(* CODESYS project IndraLogic.project

Project tree, tasks and I/O mapping:
  IndraMotionMlc1 : IndraControl XM2, Bosch Rexroth AG, order no. dependent on customer specific configuration, version 14.18.31.0
    application Application
      libraries: ML_TechBase, 14.18.0.0 (System); VisuDialogs, * (System)
      task SCC_Task (externalevent, external event EVENT_OP_MODE_MOTION_CYCLIC, priority 3, watchdog 1000 µs x 2) calls SCC, VCC, HMI
      task Acc_Sensor_Task (cyclic, interval t#2ms, priority 6) calls Acc_Sensor
      function CheckBounds [ST]
      global variables GV
      Symbols
      program VCC [FBD]
      program SCC [FBD]
      global variables MlcVarGlobal
      trace Trace (task MotionTask): VCC_Testing.uPF
      global variables UDP_Send
      function block VCC_StepFunction_Test [ST]
      trace Controller (task MotionTask): UDP_Send.Vel_RefGen, UDP_Send.Pos_RefGen, UDP_Send.nRef
      function block StepFunction_Test_Christian [ST]
      function block Input_Signals [FBD]
      function block Real_Time_Counter [FBD]
      function block Enable_Motion_SCC [FBD]
      function block JoyStick_SCC [FBD]
      function block LoadHolding_Control [FBD]
      function block JoyStick_VCC [FBD]
      function block Enable_Motion_VCC [FBD]
      function block VCC_PI_Controller [ST]
      program HMI [FBD]
      function block CyclSercosChnl [FBD]
      function block SinuousCurve_Test [ST]
      function block Ramp_Test [ST]
      function block CC_PI_FF_AD [ST]
      program VCC_Controller [FBD]
      function block VCC_Joystick_vel_ref [FBD]
      function block FIR_FIlter [ST]
      function block Discrete_FIlter [ST]
      program VCC_Testing [FBD]
      function block SCC_Controller [FBD]
      program VCC_Anti_DB [FBD]
      function block VCC_Anti_Dead_Band_v2 [ST]
      function block Subsystem [ST]
      function block VCC_SP_Ramp_Generator [ST]
      function block VCC_Controller_FF_PI_AD [ST]
      function block S_shape_Profile_old [ST]
      function block Ramp_Profile [ST]
      function block SCC_Controller_FF_PI_AD [ST]
      function block VCC_Controller_FF_PI_AD_v04 [ST]
      function block VCC_Controller_FF_PI_AD_v05 [ST]
      program VCC_PRV_Control [FBD]
      function block VCC_PRV_Mapping [ST]
      function block Discrete_Lowpass_Filter0 [ST]
      function block VCC_PV_Controller [ST]
      function block VCC_StepFunction [ST]
      function block VCC_Step_Function_Validation [ST]
      function block PF2 [ST]
      function block PF1 [ST]
      function block SCC_LPPF [ST]
      function block HPPF_pB [ST]
      function block HPPF2_pB [ST]
      function block HPPF_pA [ST]
      function block HPPF2_pA [ST]
      function block VCC_Controller_PI_FF [ST]
      function block Step_Damiano [ST]
      function block SCC_Ramp_Test [ST]
      function block SCC_HPPF [ST]
      function block SCC_DPF [ST]
      function block ZCFCN_d_FALLING [ST]
      function block ZCFCN_d_ANY [ST]
      function block SCC_Controller_VFF [ST]
      function block SCC_Controller_PFB [ST]
      function block Low_Pass_Filter [ST]
      function block SCC_PFB_Controller_PID [ST]
      function block SCC_PFB_Controller_PID2 [ST]
      function block SCC_SinProfile [ST]
      function block CascadedControllerFilter [ST]
      function block LHV_Controller [ST]
      function block LHV_Enabler [ST]
      function block Pressure_Feed_Forward [ST]
      function block SCC_Controller_PFB1 [ST]
      function block SCC_Vel_AD [ST]
      function block SCC_VFF [ST]
      function block SCC_HPPF1 [ST]
      function block LHV_Controller2 [ST]
      function block Delay_Vel [ST]
      function block Delay_Pos [ST]
      function block VCC_Controller_PFB [ST]
      function block VCC_VFF [ST]
      function block VCC_Pos_Step [ST]
      function block SCC_AD_Iq [ST]
      function block S_shape_Profile [ST]
      global variables UDP_Send_Acc
      program Acc_Sensor [FBD]
      function block SCC_Secondary_Controller [FBD]
      function block SCC_Primary_Controller [FBD]
      function block Primary_Control2 [ST]
      function block Primary_Control1 [ST]
      function block Primary_Control3 [ST]
      function block Secondary_Control [ST]
      function block LPF [ST]
      function block JoyStick_SCC_TrqCntrl [FBD]
      Visualization/
        SCC/
          visualisation SCC
          SubWindows/
            visualisation SCC_Main
            visualisation SCC_activeDamping
        VCC/
          visualisation VCC_Visualization
          visualisation VCC_Filtered_LS
          SubWindows/
      function block SCC_Acceleration_Feedback [ST]
    S20_I_O : S20_I_O, Bosch Rexroth AG, version 14.18.20.0
      S20_AI_8 : S20-AI-8, Bosch Rexroth AG, order no. R911172536, version Revision=16#0
          settings: Analog Input.IDN = 16#010005E1; Analog Input.IDN = 16#010005E1; PropritaryParameterSet_P-1-0128.0.0.IDN = 16#01009080; PropritaryParameterSet_P-1-0128.0.0.Abort if error = False; PropritaryParameterSet_P-1-0128.0.0.Jump to line if error = False; PropritaryParameterSet_P-1-0128.0.0.SercosAttribute = 16#00000000
          input  CylPos : WORD  // Analog Input.Analog Input 1
          input  p1 : WORD  // Analog Input.Analog Input 2
          input  p2 : WORD  // Analog Input.Analog Input 3
          input  p3 : WORD  // Analog Input.Analog Input 4
          input  p4 : WORD  // Analog Input.Analog Input 5
          input  p5 : WORD  // Analog Input.Analog Input 6
          input  p6 : WORD  // Analog Input.Analog Input 7
          input  p7 : WORD  // Analog Input.Analog Input 8
          unmapped channels: Analog Input
      S20_AI_8_1 : S20-AI-8, Bosch Rexroth AG, order no. R911172536, version Revision=16#0
          settings: Analog Input.IDN = 16#010005E1; Analog Input.IDN = 16#010005E1; PropritaryParameterSet_P-1-0128.0.0.IDN = 16#01009080; PropritaryParameterSet_P-1-0128.0.0.Abort if error = False; PropritaryParameterSet_P-1-0128.0.0.Jump to line if error = False; PropritaryParameterSet_P-1-0128.0.0.SercosAttribute = 16#00000000
          input  p8 : WORD  // Analog Input.Analog Input 1
          input  p9 : WORD  // Analog Input.Analog Input 2
          input  p10 : WORD  // Analog Input.Analog Input 3
          input  p11 : WORD  // Analog Input.Analog Input 4
          input  T11 : WORD  // Analog Input.Analog Input 5
          input  T6 : WORD  // Analog Input.Analog Input 6
          input  T4 : WORD  // Analog Input.Analog Input 7
          input  Acc_Y_raw : WORD  // Analog Input.Analog Input 8
          unmapped channels: Analog Input
      S20_AI_8_2 : S20-AI-8, Bosch Rexroth AG, order no. R911172536, version Revision=16#0
          settings: Analog Input.IDN = 16#010005E1; Analog Input.IDN = 16#010005E1; PropritaryParameterSet_P-1-0128.0.0.IDN = 16#01009080; PropritaryParameterSet_P-1-0128.0.0.Abort if error = False; PropritaryParameterSet_P-1-0128.0.0.Jump to line if error = False; PropritaryParameterSet_P-1-0128.0.0.SercosAttribute = 16#00000000
          input  p_pump : WORD  // Analog Input.Analog Input 1
          input  p_return : WORD  // Analog Input.Analog Input 2
          input  p_compensator : WORD  // Analog Input.Analog Input 3
          input  p_A : WORD  // Analog Input.Analog Input 4
          input  p_A1 : WORD  // Analog Input.Analog Input 5
          input  p_B : WORD  // Analog Input.Analog Input 6
          input  Q_B : WORD  // Analog Input.Analog Input 7
          input  JoyY : WORD  // Analog Input.Analog Input 8
          unmapped channels: Analog Input
      S20_AI6_AO2_SSI2 : S20-AI6-AO2-SSI2, Bosch Rexroth AG, order no. R911173120, version Revision=16#0
          settings: Analog Output.IDN = 16#010005E0; Analog Input.IDN = 16#010005E1; Positioning.IDN = 16#010005EB; Analog Output.IDN = 16#010005E0; Analog Input.IDN = 16#010005E1; Positioning.IDN = 16#010005EB; PropritaryParameterSet_P-1-0041.0.0.IDN = 16#01009029; PropritaryParameterSet_P-1-0041.0.0.Abort if error = False; PropritaryParameterSet_P-1-0041.0.0.Jump to line if error = False; PropritaryParameterSet_P-1-0041.0.0.SercosAttribute = 16#00000000; PropritaryParameterSet_P-1-0128.0.0.IDN = 16#01009080; PropritaryParameterSet_P-1-0128.0.0.Abort if error = False; PropritaryParameterSet_P-1-0128.0.0.Jump to line if error = False; PropritaryParameterSet_P-1-0128.0.0.SercosAttribute = 16#00000000; PropritaryParameterSet_P-1-0128.0.0 = [16#02,16#00,16#02,16#00,16#05,16#05]; PropritaryParameterSet_S-0-1504.0.2.IDN = 16#010205E0; PropritaryParameterSet_S-0-1504.0.2.Abort if error = False; PropritaryParameterSet_S-0-1504.0.2.Jump to line if error = False; PropritaryParameterSet_S-0-1504.0.2.SercosAttribute = 16#00000000; PropritaryParameterSet_P-1-0047.0.0.IDN = 16#0100902F; PropritaryParameterSet_P-1-0047.0.0.Abort if error = False; PropritaryParameterSet_P-1-0047.0.0.Jump to line if error = False; PropritaryParameterSet_P-1-0047.0.0.SercosAttribute = 16#00000000; PropritaryParameterSet_P-1-0128.0.1.IDN = 16#01019080; PropritaryParameterSet_P-1-0128.0.1.Abort if error = False; PropritaryParameterSet_P-1-0128.0.1.Jump to line if error = False; PropritaryParameterSet_P-1-0128.0.1.SercosAttribute = 16#00000000; PropritaryParameterSet_P-1-0128.0.1 = [16#0C,16#00,16#0C,16#00,16#05,16#05,16#0F,16#00,16#00,16#00,16#0F,16#0F,16#0F,16#00,16#00,16#00]; PropritaryParameterSet_P-1-0128.0.2.IDN = 16#01029080; PropritaryParameterSet_P-1-0128.0.2.Abort if error = False; PropritaryParameterSet_P-1-0128.0.2.Jump to line if error = False; PropritaryParameterSet_P-1-0128.0.2.SercosAttribute = 16#00000000; PropritaryParameterSet_P-1-0128.0.3.IDN = 16#01039080; PropritaryParameterSet_P-1-0128.0.3.Abort if error = False; PropritaryParameterSet_P-1-0128.0.3.Jump to line if error = False; PropritaryParameterSet_P-1-0128.0.3.SercosAttribute = 16#00000000; PropritaryParameterSet_P-1-0129.0.0.IDN = 16#01009081; PropritaryParameterSet_P-1-0129.0.0.Abort if error = False; PropritaryParameterSet_P-1-0129.0.0.Jump to line if error = False; PropritaryParameterSet_P-1-0129.0.0.SercosAttribute = 16#00000000;
            PropritaryParameterSet_P-1-0129.0.1.IDN = 16#01019081; PropritaryParameterSet_P-1-0129.0.1.Abort if error = False; PropritaryParameterSet_P-1-0129.0.1.Jump to line if error = False; PropritaryParameterSet_P-1-0129.0.1.SercosAttribute = 16#00000000; PropritaryParameterSet_P-1-0041.0.0.IDN = 16#01009029; PropritaryParameterSet_P-1-0041.0.0.Abort if error = False; PropritaryParameterSet_P-1-0041.0.0.Jump to line if error = False; PropritaryParameterSet_P-1-0041.0.0.SercosAttribute = 16#00000000
          output PVG_Us : WORD  // Analog Output.Analog Output 1
          output PRV_Cmd : WORD  // Analog Output.Analog Output 2
          input  PVG_SP : WORD  // Analog Input.Analog Input1
          input  PRV_Act : WORD  // Analog Input.Analog Input2
          unmapped channels: Analog Output, Analog Input, Positioning
      S20_DI_16_4 : S20-DI-16/4, Bosch Rexroth AG, order no. R911172532, version Revision=16#0
          settings: Digital Input.IDN = 16#010005DF; Digital Input.IDN = 16#010005DF; PropritaryParameterSet_S-0-1503.0.20.IDN = 16#011405DF
          input  startBtn : BOOL  // Digital Input.Digital Input Byte 0.00
          input  stopBtn : BOOL  // Digital Input.Digital Input Byte 0.01
          input  manMode : BOOL  // Digital Input.Digital Input Byte 0.02
          input  autoMode : BOOL  // Digital Input.Digital Input Byte 0.03
          unmapped channels: Digital Input
      S20_DO_16_3 : S20-DO-16/3, Bosch Rexroth AG, order no. R911172534, version Revision=16#0
          settings: Digital Output.IDN = 16#010005DE; Digital Output.IDN = 16#010005DE; PropritaryParameterSet_S-0-1502.0.2.IDN = 16#010205DE; PropritaryParameterSet_S-0-1502.0.20.IDN = 16#011405DE
          output LHvalve : BOOL  // Digital Output.Digital Output Byte 0.00
          output Motion_Start_Light : BOOL  // Digital Output.Digital Output Byte 0.01
          output Motion_Stop_Light : BOOL  // Digital Output.Digital Output Byte 0.02
          output CoolerFan : BOOL  // Digital Output.Digital Output Byte 0.03
          output PVG_Udc : BOOL  // Digital Output.Digital Output Byte 0.04
          unmapped channels: Digital Output
    Sercos_III_Master : SercosIII Master, Rexroth, order no. 1, version 14.6.0.0
    RT_Ethernet_Slave_XFE01_1_FB_04 : RT-Ethernet Slave(XFE01.1-FB-04), Bosch Rexroth AG, order no. R911173937, version 14.14.0.0
      Not_Used : Not Used, Bosch Rexroth AG, version 14.8.0.0
    EtherNet_IP_Adapter_on_Eng_Port : EtherNet/IP Adapter on Eng.-Port, Bosch Rexroth AG, version 12.10.2.0
      _8_Byte_Input : 8 Byte Input, Bosch Rexroth AG, version 12.10.2.0
          unmapped channels: Channel1
      _8_Byte_Output_4Byte_Run_Header : 8 Byte Output + 4Byte Run Header, Bosch Rexroth AG, version 12.10.2.0
          unmapped channels: Channel1
  libraries: VisuSymbols, 3.5.8.0 (System)
  text list GlobalTextList
*)

// IndraMotionMlc1/Application/GV

VAR_GLOBAL
	TestMode: BOOL;

	UDP_ON: BOOL;
	SCC_ON: BOOL := 0;
	SCC_On_Light: BOOL;
	SCC_ManModeVelAct: BOOL;
	SCC_AutoModeVelAct: BOOL;
	SCC_Motion_Stop_Light: BOOL;
	SCC_Manual_Mode_Enable: BOOL;
	SCC_Manual_Max_Speed: REAL := 1000.0;
	SCC_Auto_Mode_Enable: BOOL;
	SCC_Control_Mode: BOOL := 0;
	SCC_Control_Mode_Enabled: BOOL;
	SCC_Cntrl_Error_Limit: LREAL := 1;
	SCC_Cntrl_s0: LREAL := 50.0;
	SCC_Cntrl_tHold_Up_Up_Up: LREAL:= 5.0;
	SCC_Cntrl_t0: LREAL := 5.0;
	SCC_Cntrl_Pos_SP: LREAL := 200.0;
	SCC_Cntrl_Vel_SP: LREAL := 50.0;
	SCC_Cntrl_k_P: LREAL := 2.7227E+04;
	SCC_Cntrl_T_I: LREAL := 3.4851E+04;
	SCC_Cntrl_k_P_AD: LREAL := 1.4125E+05;
	SCC_Cntrl_T_I_AD: LREAL := 1.2204E+05;
	SCC_Tuning_Mode: BOOL := 0;
	SCC_S_shape_On: BOOL :=1;
	SCC_Vel_Ref_Max: REAL := 120;
	SCC_k_AD: LREAL := 2.112E-11 ;
	SCC_tau_AD: LREAL := 0.993;
	SCC_Cntrl_Motion_Cycle_Time: LREAL;
    SCC_Test_Mode: BOOL := 0; 
	SCC_Test_Mode_Enabled: BOOL := 0; 
	SCC_FB_Cntr_On: BOOL;
	SCC_FB_Cntr_Enabled: BOOL;
	SCC_I_Cntr_On: BOOL :=0;
	SCC_AD_On: BOOL :=0;
	SCC_LH_Valve_Activated: BOOL; 
	SCC_Passive_LH_On: BOOL; 
	SCC_Cntrl_FF_On: BOOL := 1;
	SCC_Cntrl_FF_up: LREAL := 1.6450e-07;
    SCC_Cntrl_FF_down: LREAL := 1.7500E-07;
	SCC_Vel_RefGen: LREAL; 
	SCC_Pos_RefGen: LREAL; 
	SCC_RecordTime: LREAL; 
	SCC_vel_AD_On: BOOL:= 0;
	SCC_vel_AD_kf: LREAL:= 1.995E04;
	SCC_vel_AD_tauf: LREAL:= 0.9934;
	SCC_HPPF_On: BOOL:= 0;
	SCC_HPPF_Reset: BOOL:= 0;
	SCC_HPPF_kf: LREAL:= 4.239E-11;
	SCC_HPPF_tauf: LREAL:= 0.999;
	SCC_LPPF_On: BOOL:= 0;
	SCC_LPPF_kf: LREAL:= 1.223E-12; 
	SCC_LPPF_tauf: LREAL:= 0.9737;
	SCC_DPF_On: BOOL:= 0;
	SCC_DPF_kf: LREAL:= 3.7255E-11;
	Joystick_Ref: LREAL; 
	SCC_OL_On: BOOL:= 0;
	SCC_Sin_Test_On: BOOL := 0;
    SCC_SinTest_T: LREAL:= 10;
	SCC_Motor_ON: BOOL := 0;
	SCC_Force_Motor_ON: BOOL := 0;
	
	SCC_LHV_OFF: BOOL := 0;
	SCC_LHV_ON: BOOL := 0;
	
	SCC_PosError_limit: LREAL:= 0.5;
	
	SCC_LHC_On: BOOL := 0;
	SCC_LHC_FF_On: BOOL := 1;
	SCC_LHC_kP: LREAL:= 0.000015;
	SCC_LHC_FF_kP: LREAL:= 0.000015;
	SCC_LHC_error_SP: LREAL:= 1;
	SCC_LHC_vel_lim: LREAL:= 0.1;
	SCC_LHC_openingDelay: TIME:= T#200MS;
	SCC_LHC_openingDelay2: TIME:= T#5MS;
	SCC_LHC_openingDelay3: TIME:= T#3S;
	SCC_Delay_ms: LREAL:= 100; 
	SCC_LHC_nSP: LREAL:= 300;
	Pos_Ref_Delay: LREAL;
	Vel_Ref_Delay: LREAL;
	Pos_Ref_Act: LREAL;
	Vel_Ref_Act: LREAL;
	SCC_Motion_Delay_On: BOOL := 0;
    SCC_Step_Test_On: BOOL := 0; 
    Mode_Selected: BOOL;
	
	SCC_AD_Iq_On: BOOL:= 0;
	SCC_k_AD_Iq: LREAL := 0 ;
	
	// Secondary Controller
	SCC_Enable_TCTR : BOOL:= 0; 
	SCC_SCTR_ON : BOOL:= 0; 
    SCC_AutoModeTorqueAct: BOOL; 
	
	// Acceleration Feedback (AF)
	SCC_AF_On: BOOL := 0;
	SCC_AF_Direct_On : BOOL := 0;
	SCC_AF_LPF_On : BOOL := 0;
	SCC_AF_LPF_w : BOOL := 0;
	SCC_AF_HPF_On : BOOL := 0;

	SCC_AF_Acc_Input_raw : LREAL;
	SCC_AF_Acc_Input : LREAL;
	SCC_AF_Acc_Input_DB : LREAL := 0.1;
	
	SCC_AF_D_rev : LREAL := 10.6;
	SCC_AF_K_direct : LREAL := 1.7045E-04;
	SCC_AF_LPF_Num1 : LREAL := 0;
	SCC_AF_LPF_Num2 : LREAL := 1.39E-05;
	SCC_AF_LPF_Den1 : LREAL := 1;
	SCC_AF_LPF_Den2 : LREAL := -0.9418;
	SCC_AF_HPF_Num1 : LREAL := 2.6846E-04;
	SCC_AF_HPF_Num2 : LREAL := -2.6846E-04;
	SCC_AF_HPF_Den1 : LREAL := 1;
	SCC_AF_HPF_Den2 : LREAL := -0.9955;

	Ramp_tHold: LREAL:= 1;
	Ramp_tWait: LREAL:= 1;
	tRamp: LREAL:= 1;
	nSP: LREAL:= 1000;
	
	VCC_ON: BOOL := 0; 
	VCC_On_Light: BOOL;
	VCC_Manual_Mode_Enabled: BOOL; 
	VCC_S_shape_On: BOOL :=1;
    VCC_Vel_Ref_Max: REAL := 120;
    VCC_Max_Joy_Output: REAL := 100.0;
    VCC_Auto_Mode_Enabled: BOOL; 
	VCC_Control_Mode: BOOL := 0;
    VCC_Control_Mode_Enabled: BOOL := 0;
	VCC_FB_Cntr_On: BOOL :=0;
	VCC_FB_Cntr_Enabled: BOOL;
	VCC_I_Cntr_On: BOOL :=0;
	VCC_AD_On: BOOL :=0;
	VCC_k_AD: LREAL := 0.004;
	VCC_Cntrl_DB_up: LREAL := 0.114;
	VCC_Cntrl_Motion_Cycle_Time: LREAL;
    VCC_Cntrl_DB_down: LREAL := 0.13;
	VCC_Cntrl_Error_Limit: LREAL := 1;
	VCC_Cntrl_s0: LREAL := 50.0;
	VCC_Cntrl_Trvl_Dist: LREAL := 200.0;
	VCC_Cntrl_tHold: LREAL:= 5.0;
	VCC_Cntrl_t0: LREAL := 3.0;
	VCC_Cntrl_Vel_SP: LREAL := 50.0;
	VCC_Cntrl_k_P: LREAL := 29.1743;
	VCC_Cntrl_T_I: LREAL := 19.4884;
	VCC_Tuning_Mode: BOOL := 0;
	VCC_Test_Mode: BOOL := 0; 
	VCC_Test_Mode_Enabled: BOOL := 0; 
	VCC_Ramp_Test_On: BOOL := 0; 
	VCC_Ramp_Test_u_DCV_1: LREAL := 0; 
	VCC_Ramp_Test_u_DCV_2: LREAL := 0; 
	VCC_Ramp_Test_tR: LREAL := 1; 
	VCC_Ramp_Test_tHold_Up: LREAL := 5; 
	VCC_Ramp_Test_tHold_Down: LREAL := 5; 
	VCC_Ramp_Test_tWait: LREAL := 5; 
	VCC_Step_Test_On: BOOL := 0; 
	VCC_Step_Test_t0: LREAL := 1;
	VCC_Step_Test_tWait: LREAL := 1;
	VCC_Step_Test_tWait2: LREAL := 1;
    VCC_Step_Test_tStepUp: LREAL := 1;
	VCC_Step_Test_tStepDown: LREAL := 1;
	VCC_Step_Test_SP: LREAL := 0.1;
	VCC_Step_Test_u0: LREAL := 0.05;
	VCC_Step_Test_Up: BOOL := 0; 
	VCC_Sin_Test_On: BOOL := 0; 
	VCC_Test_t0: LREAL := 1.0;
	VCC_Vel_RefGen: LREAL; 
	VCC_Pos_RefGen: LREAL; 
	VCC_RecordTime: LREAL; 
	VCC_Cntrl_Q_max_up: LREAL := 30.0;
	VCC_Cntrl_Q_max_down: LREAL := 30.0;
	VCC_Cntrl_FF_Valve_Mapping_On: BOOL := 0; 
	VCC_Cntrl_Integral_Reset_On: BOOL := 1; 
	VCC_PRV_Cntrl_p_C_Max: LREAL := 75; 
	VCC_PRV_Cntrl_p_C_Min: LREAL := 4; 
	VCC_PRV_Cntrl_Opening: LREAL := 0;
	VCC_PRV_Cntrl_Opening_SP: LREAL := 0;
	VCC_PRV_Cntrl_Enable: BOOL := 0;
	VCC_PRV_Cntrl_Enabled: BOOL;
	VCC_PRV_Cntrl_Auto_On: BOOL := 0;
	VCC_PRV_p_C_SP: LREAL := 0;
	VCC_PRV_Cntrl_Manual_Pressure_On: BOOL;
	VCC_PRV_Cntrl_k_LPF: LREAL :=1;
	VCC_PRV_Cntrl_T_LPF: LREAL :=0.5;
	VCC_PRV_Cntrl_k_P: LREAL := 1; 
	VCC_PRV_Cntrl_T_I: LREAL := 0; 
	VCC_PRV_Cntrl_FF_On: BOOL := 1; 
	VCC_PRV_Cntrl_LPF_On: BOOL := 1; 
	VCC_PRV_Cntrl_Tuning_Mode_On: BOOL := 0; 
	VCC_PF2_On: BOOL := 0; 
	VCC_PF1_On: BOOL := 0; 
    VCC_PF_pB_On: BOOL := 0; 
	VCC_PF_pB_vInv_On: BOOL := 0; 
	VCC_PF_pA_vInv_On: BOOL := 0; 
	VCC_PF_pL_vInv_On: BOOL := 0; 
	VCC_PF_Test_On: BOOL := 0; 
	VCC_PF_HP_Num1: LREAL := 1.176E-11;  
	VCC_PF_HP_Den1: LREAL := 1;
	VCC_PF_HP_Den2: LREAL := -0.9957;
	VCC_PF1_HP_Num1: LREAL := 9.019E-12;  
	VCC_PF1_HP_Den1: LREAL := 1;
	VCC_PF1_HP_Den2: LREAL := -0.9905;
	VCC_PF_pB_HP_Num1: LREAL := 1.344E-11;  
	VCC_PF_pB_HP_Den1: LREAL := 1;
	VCC_PF_pB_HP_Den2: LREAL := -0.9951;
	VCC_PF_ADB_On: BOOL := 0; 
	VCC_LPPF_On: BOOL := 0; 
	VCC_LPPF_Num1: LREAL := 8.647E-13;  
	VCC_LPPF_Den1: LREAL := 1;
	VCC_LPPF_Den2: LREAL := -0.8424;
	VCC_SinTest_freq: LREAL := 0;
	VCC_SinTest_Amp: LREAL := 0;
	VCC_Cntrl_uPF: LREAL := 0;
END_VAR

// IndraMotionMlc1/Application/MlcVarGlobal
(* Automatically generated code by XLC/MLC. *)
(* Please don't edit, the code will be overwritten. For usercode use UserVarGlobal! *)
{attribute 'linkalways'}
{attribute 'analysis' := '-33'}
VAR_GLOBAL CONSTANT

(*LREAL axis "Drive1" with axis number 1*)
Drive1: AXIS_REF :=(CntrlNo:=LOCAL_CNTRL,AxisNo:=AXIS_1);


(*Probe 001*)
TouchProbe001: TOUCHPROBE_REF :=(CntrlNo:=LOCAL_CNTRL,TouchProbeNo:=TOUCHPROBE_1);

(*Probe 002*)
TouchProbe002: TOUCHPROBE_REF :=(CntrlNo:=LOCAL_CNTRL,TouchProbeNo:=TOUCHPROBE_2);

(*Probe 003*)
TouchProbe003: TOUCHPROBE_REF :=(CntrlNo:=LOCAL_CNTRL,TouchProbeNo:=TOUCHPROBE_3);

(*Probe 004*)
TouchProbe004: TOUCHPROBE_REF :=(CntrlNo:=LOCAL_CNTRL,TouchProbeNo:=TOUCHPROBE_4);

(*Probe 005*)
TouchProbe005: TOUCHPROBE_REF :=(CntrlNo:=LOCAL_CNTRL,TouchProbeNo:=TOUCHPROBE_5);

(*Probe 006*)
TouchProbe006: TOUCHPROBE_REF :=(CntrlNo:=LOCAL_CNTRL,TouchProbeNo:=TOUCHPROBE_6);

(*Probe 007*)
TouchProbe007: TOUCHPROBE_REF :=(CntrlNo:=LOCAL_CNTRL,TouchProbeNo:=TOUCHPROBE_7);

(*Probe 008*)
TouchProbe008: TOUCHPROBE_REF :=(CntrlNo:=LOCAL_CNTRL,TouchProbeNo:=TOUCHPROBE_8);

(*Probe 009*)
TouchProbe009: TOUCHPROBE_REF :=(CntrlNo:=LOCAL_CNTRL,TouchProbeNo:=TOUCHPROBE_9);

(*Probe 010*)
TouchProbe010: TOUCHPROBE_REF :=(CntrlNo:=LOCAL_CNTRL,TouchProbeNo:=TOUCHPROBE_10);

(*Probe 011*)
TouchProbe011: TOUCHPROBE_REF :=(CntrlNo:=LOCAL_CNTRL,TouchProbeNo:=TOUCHPROBE_11);

(*Probe 012*)
TouchProbe012: TOUCHPROBE_REF :=(CntrlNo:=LOCAL_CNTRL,TouchProbeNo:=TOUCHPROBE_12);

(*Probe 013*)
TouchProbe013: TOUCHPROBE_REF :=(CntrlNo:=LOCAL_CNTRL,TouchProbeNo:=TOUCHPROBE_13);

(*Probe 014*)
TouchProbe014: TOUCHPROBE_REF :=(CntrlNo:=LOCAL_CNTRL,TouchProbeNo:=TOUCHPROBE_14);

(*Probe 015*)
TouchProbe015: TOUCHPROBE_REF :=(CntrlNo:=LOCAL_CNTRL,TouchProbeNo:=TOUCHPROBE_15);

(*Probe 016*)
TouchProbe016: TOUCHPROBE_REF :=(CntrlNo:=LOCAL_CNTRL,TouchProbeNo:=TOUCHPROBE_16);

(*Probe 017*)
TouchProbe017: TOUCHPROBE_REF :=(CntrlNo:=LOCAL_CNTRL,TouchProbeNo:=TOUCHPROBE_17);

(*Probe 018*)
TouchProbe018: TOUCHPROBE_REF :=(CntrlNo:=LOCAL_CNTRL,TouchProbeNo:=TOUCHPROBE_18);

(*Probe 019*)
TouchProbe019: TOUCHPROBE_REF :=(CntrlNo:=LOCAL_CNTRL,TouchProbeNo:=TOUCHPROBE_19);

(*Probe 020*)
TouchProbe020: TOUCHPROBE_REF :=(CntrlNo:=LOCAL_CNTRL,TouchProbeNo:=TOUCHPROBE_20);

(*Probe 021*)
TouchProbe021: TOUCHPROBE_REF :=(CntrlNo:=LOCAL_CNTRL,TouchProbeNo:=TOUCHPROBE_21);

(*Probe 022*)
TouchProbe022: TOUCHPROBE_REF :=(CntrlNo:=LOCAL_CNTRL,TouchProbeNo:=TOUCHPROBE_22);

(*Probe 023*)
TouchProbe023: TOUCHPROBE_REF :=(CntrlNo:=LOCAL_CNTRL,TouchProbeNo:=TOUCHPROBE_23);

(*Probe 024*)
TouchProbe024: TOUCHPROBE_REF :=(CntrlNo:=LOCAL_CNTRL,TouchProbeNo:=TOUCHPROBE_24);

(*Probe 025*)
TouchProbe025: TOUCHPROBE_REF :=(CntrlNo:=LOCAL_CNTRL,TouchProbeNo:=TOUCHPROBE_25);

(*Probe 026*)
TouchProbe026: TOUCHPROBE_REF :=(CntrlNo:=LOCAL_CNTRL,TouchProbeNo:=TOUCHPROBE_26);

(*Probe 027*)
TouchProbe027: TOUCHPROBE_REF :=(CntrlNo:=LOCAL_CNTRL,TouchProbeNo:=TOUCHPROBE_27);

(*Probe 028*)
TouchProbe028: TOUCHPROBE_REF :=(CntrlNo:=LOCAL_CNTRL,TouchProbeNo:=TOUCHPROBE_28);

(*Probe 029*)
TouchProbe029: TOUCHPROBE_REF :=(CntrlNo:=LOCAL_CNTRL,TouchProbeNo:=TOUCHPROBE_29);

(*Probe 030*)
TouchProbe030: TOUCHPROBE_REF :=(CntrlNo:=LOCAL_CNTRL,TouchProbeNo:=TOUCHPROBE_30);

(*Probe 031*)
TouchProbe031: TOUCHPROBE_REF :=(CntrlNo:=LOCAL_CNTRL,TouchProbeNo:=TOUCHPROBE_31);

(*Probe 032*)
TouchProbe032: TOUCHPROBE_REF :=(CntrlNo:=LOCAL_CNTRL,TouchProbeNo:=TOUCHPROBE_32);

(*Probe 033*)
TouchProbe033: TOUCHPROBE_REF :=(CntrlNo:=LOCAL_CNTRL,TouchProbeNo:=TOUCHPROBE_33);

(*Probe 034*)
TouchProbe034: TOUCHPROBE_REF :=(CntrlNo:=LOCAL_CNTRL,TouchProbeNo:=TOUCHPROBE_34);

(*Probe 035*)
TouchProbe035: TOUCHPROBE_REF :=(CntrlNo:=LOCAL_CNTRL,TouchProbeNo:=TOUCHPROBE_35);

(*Probe 036*)
TouchProbe036: TOUCHPROBE_REF :=(CntrlNo:=LOCAL_CNTRL,TouchProbeNo:=TOUCHPROBE_36);

(*Probe 037*)
TouchProbe037: TOUCHPROBE_REF :=(CntrlNo:=LOCAL_CNTRL,TouchProbeNo:=TOUCHPROBE_37);

(*Probe 038*)
TouchProbe038: TOUCHPROBE_REF :=(CntrlNo:=LOCAL_CNTRL,TouchProbeNo:=TOUCHPROBE_38);

(*Probe 039*)
TouchProbe039: TOUCHPROBE_REF :=(CntrlNo:=LOCAL_CNTRL,TouchProbeNo:=TOUCHPROBE_39);

(*Probe 040*)
TouchProbe040: TOUCHPROBE_REF :=(CntrlNo:=LOCAL_CNTRL,TouchProbeNo:=TOUCHPROBE_40);

(*Probe 041*)
TouchProbe041: TOUCHPROBE_REF :=(CntrlNo:=LOCAL_CNTRL,TouchProbeNo:=TOUCHPROBE_41);

(*Probe 042*)
TouchProbe042: TOUCHPROBE_REF :=(CntrlNo:=LOCAL_CNTRL,TouchProbeNo:=TOUCHPROBE_42);

(*Probe 043*)
TouchProbe043: TOUCHPROBE_REF :=(CntrlNo:=LOCAL_CNTRL,TouchProbeNo:=TOUCHPROBE_43);

(*Probe 044*)
TouchProbe044: TOUCHPROBE_REF :=(CntrlNo:=LOCAL_CNTRL,TouchProbeNo:=TOUCHPROBE_44);

(*Probe 045*)
TouchProbe045: TOUCHPROBE_REF :=(CntrlNo:=LOCAL_CNTRL,TouchProbeNo:=TOUCHPROBE_45);

(*Probe 046*)
TouchProbe046: TOUCHPROBE_REF :=(CntrlNo:=LOCAL_CNTRL,TouchProbeNo:=TOUCHPROBE_46);

(*Probe 047*)
TouchProbe047: TOUCHPROBE_REF :=(CntrlNo:=LOCAL_CNTRL,TouchProbeNo:=TOUCHPROBE_47);

(*Probe 048*)
TouchProbe048: TOUCHPROBE_REF :=(CntrlNo:=LOCAL_CNTRL,TouchProbeNo:=TOUCHPROBE_48);

(*Probe 049*)
TouchProbe049: TOUCHPROBE_REF :=(CntrlNo:=LOCAL_CNTRL,TouchProbeNo:=TOUCHPROBE_49);

(*Probe 050*)
TouchProbe050: TOUCHPROBE_REF :=(CntrlNo:=LOCAL_CNTRL,TouchProbeNo:=TOUCHPROBE_50);

(*Probe 051*)
TouchProbe051: TOUCHPROBE_REF :=(CntrlNo:=LOCAL_CNTRL,TouchProbeNo:=TOUCHPROBE_51);

(*Probe 052*)
TouchProbe052: TOUCHPROBE_REF :=(CntrlNo:=LOCAL_CNTRL,TouchProbeNo:=TOUCHPROBE_52);

(*Probe 053*)
TouchProbe053: TOUCHPROBE_REF :=(CntrlNo:=LOCAL_CNTRL,TouchProbeNo:=TOUCHPROBE_53);

(*Probe 054*)
TouchProbe054: TOUCHPROBE_REF :=(CntrlNo:=LOCAL_CNTRL,TouchProbeNo:=TOUCHPROBE_54);

(*Probe 055*)
TouchProbe055: TOUCHPROBE_REF :=(CntrlNo:=LOCAL_CNTRL,TouchProbeNo:=TOUCHPROBE_55);

(*Probe 056*)
TouchProbe056: TOUCHPROBE_REF :=(CntrlNo:=LOCAL_CNTRL,TouchProbeNo:=TOUCHPROBE_56);

(*Probe 057*)
TouchProbe057: TOUCHPROBE_REF :=(CntrlNo:=LOCAL_CNTRL,TouchProbeNo:=TOUCHPROBE_57);

(*Probe 058*)
TouchProbe058: TOUCHPROBE_REF :=(CntrlNo:=LOCAL_CNTRL,TouchProbeNo:=TOUCHPROBE_58);

(*Probe 059*)
TouchProbe059: TOUCHPROBE_REF :=(CntrlNo:=LOCAL_CNTRL,TouchProbeNo:=TOUCHPROBE_59);

(*Probe 060*)
TouchProbe060: TOUCHPROBE_REF :=(CntrlNo:=LOCAL_CNTRL,TouchProbeNo:=TOUCHPROBE_60);

(*Probe 061*)
TouchProbe061: TOUCHPROBE_REF :=(CntrlNo:=LOCAL_CNTRL,TouchProbeNo:=TOUCHPROBE_61);

(*Probe 062*)
TouchProbe062: TOUCHPROBE_REF :=(CntrlNo:=LOCAL_CNTRL,TouchProbeNo:=TOUCHPROBE_62);

(*Probe 063*)
TouchProbe063: TOUCHPROBE_REF :=(CntrlNo:=LOCAL_CNTRL,TouchProbeNo:=TOUCHPROBE_63);

(*Probe 064*)
TouchProbe064: TOUCHPROBE_REF :=(CntrlNo:=LOCAL_CNTRL,TouchProbeNo:=TOUCHPROBE_64);

(*Probe 065*)
TouchProbe065: TOUCHPROBE_REF :=(CntrlNo:=LOCAL_CNTRL,TouchProbeNo:=TOUCHPROBE_65);

(*Probe 066*)
TouchProbe066: TOUCHPROBE_REF :=(CntrlNo:=LOCAL_CNTRL,TouchProbeNo:=TOUCHPROBE_66);

(*Probe 067*)
TouchProbe067: TOUCHPROBE_REF :=(CntrlNo:=LOCAL_CNTRL,TouchProbeNo:=TOUCHPROBE_67);

(*Probe 068*)
TouchProbe068: TOUCHPROBE_REF :=(CntrlNo:=LOCAL_CNTRL,TouchProbeNo:=TOUCHPROBE_68);

(*Probe 069*)
TouchProbe069: TOUCHPROBE_REF :=(CntrlNo:=LOCAL_CNTRL,TouchProbeNo:=TOUCHPROBE_69);

(*Probe 070*)
TouchProbe070: TOUCHPROBE_REF :=(CntrlNo:=LOCAL_CNTRL,TouchProbeNo:=TOUCHPROBE_70);

(*Probe 071*)
TouchProbe071: TOUCHPROBE_REF :=(CntrlNo:=LOCAL_CNTRL,TouchProbeNo:=TOUCHPROBE_71);

(*Probe 072*)
TouchProbe072: TOUCHPROBE_REF :=(CntrlNo:=LOCAL_CNTRL,TouchProbeNo:=TOUCHPROBE_72);

(*Probe 073*)
TouchProbe073: TOUCHPROBE_REF :=(CntrlNo:=LOCAL_CNTRL,TouchProbeNo:=TOUCHPROBE_73);

(*Probe 074*)
TouchProbe074: TOUCHPROBE_REF :=(CntrlNo:=LOCAL_CNTRL,TouchProbeNo:=TOUCHPROBE_74);

(*Probe 075*)
TouchProbe075: TOUCHPROBE_REF :=(CntrlNo:=LOCAL_CNTRL,TouchProbeNo:=TOUCHPROBE_75);

(*Probe 076*)
TouchProbe076: TOUCHPROBE_REF :=(CntrlNo:=LOCAL_CNTRL,TouchProbeNo:=TOUCHPROBE_76);

(*Probe 077*)
TouchProbe077: TOUCHPROBE_REF :=(CntrlNo:=LOCAL_CNTRL,TouchProbeNo:=TOUCHPROBE_77);

(*Probe 078*)
TouchProbe078: TOUCHPROBE_REF :=(CntrlNo:=LOCAL_CNTRL,TouchProbeNo:=TOUCHPROBE_78);

(*Probe 079*)
TouchProbe079: TOUCHPROBE_REF :=(CntrlNo:=LOCAL_CNTRL,TouchProbeNo:=TOUCHPROBE_79);

(*Probe 080*)
TouchProbe080: TOUCHPROBE_REF :=(CntrlNo:=LOCAL_CNTRL,TouchProbeNo:=TOUCHPROBE_80);

(*Probe 081*)
TouchProbe081: TOUCHPROBE_REF :=(CntrlNo:=LOCAL_CNTRL,TouchProbeNo:=TOUCHPROBE_81);

(*Probe 082*)
TouchProbe082: TOUCHPROBE_REF :=(CntrlNo:=LOCAL_CNTRL,TouchProbeNo:=TOUCHPROBE_82);

(*Probe 083*)
TouchProbe083: TOUCHPROBE_REF :=(CntrlNo:=LOCAL_CNTRL,TouchProbeNo:=TOUCHPROBE_83);

(*Probe 084*)
TouchProbe084: TOUCHPROBE_REF :=(CntrlNo:=LOCAL_CNTRL,TouchProbeNo:=TOUCHPROBE_84);

(*Probe 085*)
TouchProbe085: TOUCHPROBE_REF :=(CntrlNo:=LOCAL_CNTRL,TouchProbeNo:=TOUCHPROBE_85);

(*Probe 086*)
TouchProbe086: TOUCHPROBE_REF :=(CntrlNo:=LOCAL_CNTRL,TouchProbeNo:=TOUCHPROBE_86);

(*Probe 087*)
TouchProbe087: TOUCHPROBE_REF :=(CntrlNo:=LOCAL_CNTRL,TouchProbeNo:=TOUCHPROBE_87);

(*Probe 088*)
TouchProbe088: TOUCHPROBE_REF :=(CntrlNo:=LOCAL_CNTRL,TouchProbeNo:=TOUCHPROBE_88);

(*Probe 089*)
TouchProbe089: TOUCHPROBE_REF :=(CntrlNo:=LOCAL_CNTRL,TouchProbeNo:=TOUCHPROBE_89);

(*Probe 090*)
TouchProbe090: TOUCHPROBE_REF :=(CntrlNo:=LOCAL_CNTRL,TouchProbeNo:=TOUCHPROBE_90);

(*Probe 091*)
TouchProbe091: TOUCHPROBE_REF :=(CntrlNo:=LOCAL_CNTRL,TouchProbeNo:=TOUCHPROBE_91);

(*Probe 092*)
TouchProbe092: TOUCHPROBE_REF :=(CntrlNo:=LOCAL_CNTRL,TouchProbeNo:=TOUCHPROBE_92);

(*Probe 093*)
TouchProbe093: TOUCHPROBE_REF :=(CntrlNo:=LOCAL_CNTRL,TouchProbeNo:=TOUCHPROBE_93);

(*Probe 094*)
TouchProbe094: TOUCHPROBE_REF :=(CntrlNo:=LOCAL_CNTRL,TouchProbeNo:=TOUCHPROBE_94);

(*Probe 095*)
TouchProbe095: TOUCHPROBE_REF :=(CntrlNo:=LOCAL_CNTRL,TouchProbeNo:=TOUCHPROBE_95);

(*Probe 096*)
TouchProbe096: TOUCHPROBE_REF :=(CntrlNo:=LOCAL_CNTRL,TouchProbeNo:=TOUCHPROBE_96);

(*Probe 097*)
TouchProbe097: TOUCHPROBE_REF :=(CntrlNo:=LOCAL_CNTRL,TouchProbeNo:=TOUCHPROBE_97);

(*Probe 098*)
TouchProbe098: TOUCHPROBE_REF :=(CntrlNo:=LOCAL_CNTRL,TouchProbeNo:=TOUCHPROBE_98);

(*Probe 099*)
TouchProbe099: TOUCHPROBE_REF :=(CntrlNo:=LOCAL_CNTRL,TouchProbeNo:=TOUCHPROBE_99);

(*Probe 100*)
TouchProbe100: TOUCHPROBE_REF :=(CntrlNo:=LOCAL_CNTRL,TouchProbeNo:=TOUCHPROBE_100);

END_VAR

// IndraMotionMlc1/Application/UDP_Send
{attribute 'qualified_only'}
VAR_GLOBAL
    plcTime : LREAL := 0.000;
	RecordTime : LREAL := 0.000;
	PwrOn : BOOL;
    LHvalve_Open: BOOL;
	ActualVel : REAL;
	InterpolVel : REAL;
	n_SP : REAL;
    Sc_DataA : REAL;
	Sc_DataB  : REAL;
	Sc_DataC  : REAL;
	Sc_DataD  : REAL;
	Sc_DataE  : REAL;
	Sc_DataF  : REAL;
	ActualTorque : REAL;
	ActualCylPos : REAL;
	Pos_RefGen : LREAL;
	Vel_RefGen : LREAL;
	AccRefGen : LREAL;
	JerkRefGen : LREAL;
	nRef : LREAL;
    p_001: REAL;
	p_002: REAL;
	p_003: REAL;
	p_004: REAL;
	p_005: REAL;
	p_006: REAL;
	p_007: REAL;
	p_008: REAL;
	p_009: REAL;
	p_010: REAL;
	p_011: REAL;
	T004: REAL;
	Acc_Y: REAL;
	T006: REAL;
	T011: REAL;
	pP: REAL;
	pR: REAL;
	pA: REAL;
	pA1: REAL;
	pB: REAL;
	pC: REAL;
	QB: REAL;
    PVG_SP: REAL; 
	VCC_Opening_Cmd: REAL; 
	VCC_uDCV_ref: REAL; 
	u_FF: REAL;
	u_P_cntr: REAL;
	u_I_cntr: REAL;
	pB_Filtered: REAL; 
	PRV_Cmd_Opening: REAL; 
	tau_emref_UDP : REAL ;
	tau_emref_sat_UDP : REAL ;
	
	(*nArray : ARRAY [0..3] OF DINT := [1, 2, 3, 4];*)
	
END_VAR

// IndraMotionMlc1/Application/UDP_Send_Acc
{attribute 'qualified_only'}
VAR_GLOBAL
	Acc_Y2 : LREAL; 
	AccRefGen2 : LREAL;
END_VAR

// IndraMotionMlc1/Application/SCC
PROGRAM SCC
VAR
	Enable_Motion_SCC_0: Enable_Motion_SCC;
	Motion_Enabled: BOOL;
   	Real_Time_Counter_0: Real_Time_Counter;
	ML_WriteCyclicVelocity_0: ML_WriteCyclicVelocity;
	GreenLight: SR;
	MB_ReadRealParameter_1: MB_ReadRealParameter;
	CyclSercosChnl_0: CyclSercosChnl;
	ML_WriteCyclicVelocity_1: ML_WriteCyclicVelocity;
	JoyStick_SCC_0: JoyStick_SCC;
	EnableCyclicVelocit1: ML_OpenCyclicVelocityChannel;
	StepFunction_Test_Christian_0: StepFunction_Test_Christian;

	LoadHolding_Control_0: LoadHolding_Control;
	n_ref: LREAL;

	s0: LREAL :=50;
	t0: LREAL :=5;
	tHold_Up_Up_Up: LREAL :=3 ;
	xTravel: LREAL := 400;
	a_SP: LREAL := 150;
	n_SP: LREAL := 150;
	MaxError: LREAL := 1.0;
	kI: LREAL;
	kP: LREAL := 30;
	LHenable: BOOL;
	Force_LH_Valve_Open: BOOL;
	SCC_Controller_0: SCC_Controller;
	SCC_Primary_Controller_0: SCC_Primary_Controller;
	ML_WriteCyclicTorque_0: ML_WriteCyclicTorque;
	Test: LREAL;
	SCC_Secondary_Controller_0: SCC_Secondary_Controller;
	tau_ref: REAL;
	test6: LREAL;
	ML_WriteCyclicTorqueCtrl_1: ML_WriteCyclicTorqueCtrl;
		JoyStick_SCC_TrqCntrl_0: JoyStick_SCC_TrqCntrl;
		MinTorque:REAL := -95;
	InitTorque:REAL := 50;
	MaxTorque:REAL := 95;
		TrqCommand: REAL;
	ML_WriteCyclicTorque_1: ML_WriteCyclicTorque;
END_VAR

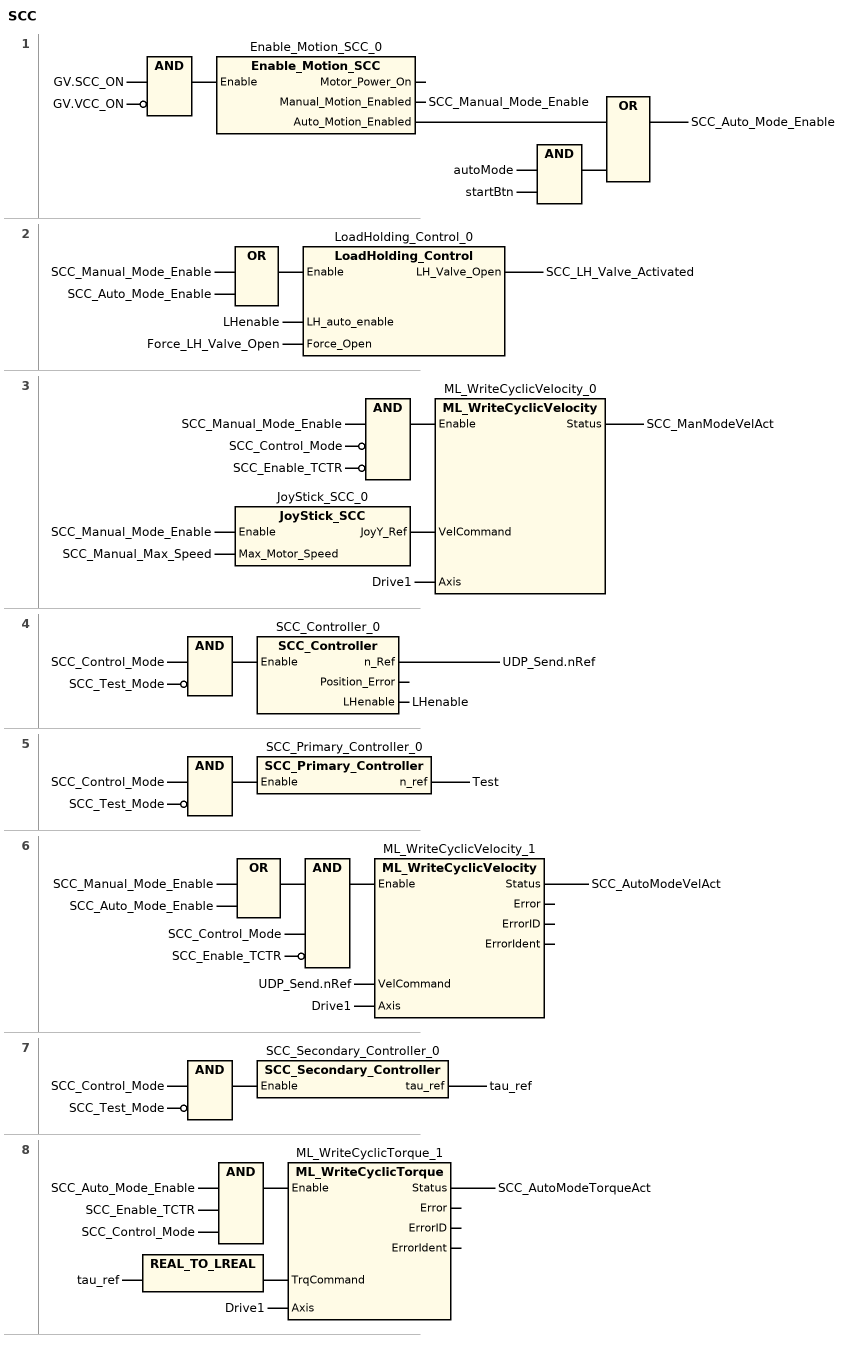
// NETWORK 1
Enable_Motion_SCC_0(Enable := GV.SCC_ON AND NOT GV.VCC_ON, Manual_Motion_Enabled => SCC_Manual_Mode_Enable); // Enable_Motion_SCC
SCC_Auto_Mode_Enable := Enable_Motion_SCC_0.Auto_Motion_Enabled OR autoMode AND startBtn;

// NETWORK 2
LoadHolding_Control_0(
    Enable := SCC_Manual_Mode_Enable OR SCC_Auto_Mode_Enable,
    LH_auto_enable := LHenable,
    Force_Open := Force_LH_Valve_Open); // LoadHolding_Control
SCC_LH_Valve_Activated := LoadHolding_Control_0.LH_Valve_Open;

// NETWORK 3
JoyStick_SCC_0(Enable := SCC_Manual_Mode_Enable, Max_Motor_Speed := SCC_Manual_Max_Speed); // JoyStick_SCC
ML_WriteCyclicVelocity_0(
    Enable := SCC_Manual_Mode_Enable AND NOT SCC_Control_Mode AND NOT SCC_Enable_TCTR,
    VelCommand := JoyStick_SCC_0.JoyY_Ref,
    Axis := Drive1); // ML_WriteCyclicVelocity
SCC_ManModeVelAct := ML_WriteCyclicVelocity_0.Status;

// NETWORK 4
SCC_Controller_0(Enable := SCC_Control_Mode AND NOT SCC_Test_Mode, LHenable => LHenable); // SCC_Controller
UDP_Send.nRef := SCC_Controller_0.n_Ref;

// NETWORK 5
SCC_Primary_Controller_0(Enable := SCC_Control_Mode AND NOT SCC_Test_Mode); // SCC_Primary_Controller
Test := SCC_Primary_Controller_0.n_ref;

// NETWORK 6
ML_WriteCyclicVelocity_1(
    Enable := (SCC_Manual_Mode_Enable OR SCC_Auto_Mode_Enable) AND SCC_Control_Mode AND NOT SCC_Enable_TCTR,
    VelCommand := UDP_Send.nRef,
    Axis := Drive1); // ML_WriteCyclicVelocity
SCC_AutoModeVelAct := ML_WriteCyclicVelocity_1.Status;

// NETWORK 7
SCC_Secondary_Controller_0(Enable := SCC_Control_Mode AND NOT SCC_Test_Mode); // SCC_Secondary_Controller
tau_ref := SCC_Secondary_Controller_0.tau_ref;

// NETWORK 8
ML_WriteCyclicTorque_1(
    Enable := SCC_Auto_Mode_Enable AND SCC_Enable_TCTR AND SCC_Control_Mode,
    TrqCommand := REAL_TO_LREAL(tau_ref),
    Axis := Drive1); // ML_WriteCyclicTorque
SCC_AutoModeTorqueAct := ML_WriteCyclicTorque_1.Status;

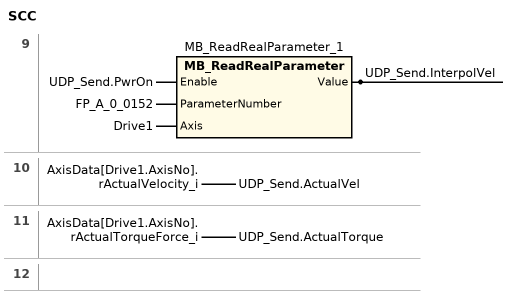
// NETWORK 9
MB_ReadRealParameter_1(
    Enable := UDP_Send.PwrOn,
    ParameterNumber := FP_A_0_0152,
    Axis := Drive1,
    Value => UDP_Send.InterpolVel); // MB_ReadRealParameter

// NETWORK 10
UDP_Send.ActualVel := AxisData[Drive1.AxisNo].rActualVelocity_i;

// NETWORK 11
UDP_Send.ActualTorque := AxisData[Drive1.AxisNo].rActualTorqueForce_i;

// NETWORK 12

END_PROGRAM

// IndraMotionMlc1/Application/Enable_Motion_SCC
FUNCTION_BLOCK Enable_Motion_SCC
VAR_INPUT
	Enable: BOOL;
END_VAR
VAR_OUTPUT
	Motor_Power_On: BOOL;
 	Manual_Motion_Enabled: BOOL;
	Auto_Motion_Enabled: BOOL;
END_VAR
VAR
	Power_On_1: RS;
	Motor_Error: BOOL;
	Motor_Power_On_0: MC_Power;
	Motor_Stop: MC_Stop;
	Motor_Stopped: BOOL;
	Real_Time_Counter_0: Real_Time_Counter;
	System_Ready: BOOL;
	MC_Reset_0: MC_Reset;
	Stopp: RS;
	TON_0: TON;
	TON_1: TON;
	TON_2: TON;
	TOF_0: TOF;
	TOF_1: TOF;
	R_TRIG_1: R_TRIG;
	GreenLight: SR;
	EnableCyclicVelocit: ML_OpenCyclicVelocityChannel;	
	EnableCyclicVelocit_1: ML_OpenCyclicVelocityChannel;
	
	R_TRIG_0: R_TRIG;
	R_TRIG_2: R_TRIG;
	F_TRIG_0: F_TRIG;
	R_TRIG_3: R_TRIG;
	R_TRIG_4: R_TRIG;
	TON_3: TON;
	ML_OpenCyclicTorqueChannel_0: ML_OpenCyclicTorqueChannel;
	VCTR_Enabled: BOOL;
	TCTR_Enabled: BOOL;
	VCTR_Manual_Enabled: BOOL;
	ML_OpenCyclicTorqueChannelCtrl_0: ML_OpenCyclicTorqueChannelCtrl;
	ML_OpenCyclicTorqueChannel_1: ML_OpenCyclicTorqueChannel;
END_VAR

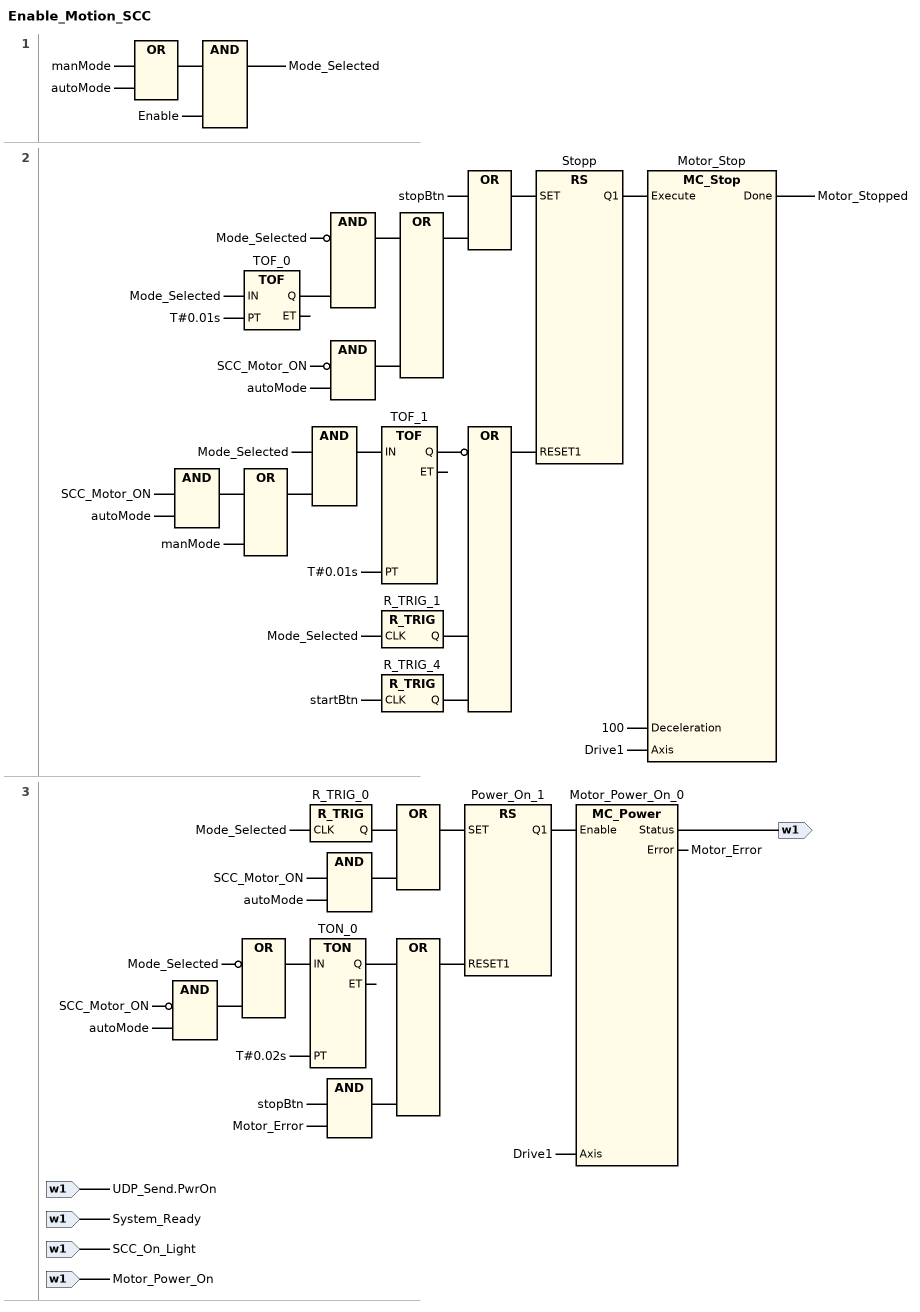
// NETWORK 1
Mode_Selected := (manMode OR autoMode) AND Enable;

// NETWORK 2
TOF_0(IN := Mode_Selected, PT := T#0.01s); // TOF
TOF_1(IN := Mode_Selected AND (SCC_Motor_ON AND autoMode OR manMode), PT := T#0.01s); // TOF
R_TRIG_1(CLK := Mode_Selected); // R_TRIG
R_TRIG_4(CLK := startBtn); // R_TRIG
Stopp(SET := stopBtn OR (NOT Mode_Selected AND TOF_0.Q OR NOT SCC_Motor_ON AND autoMode), RESET1 := NOT TOF_1.Q OR R_TRIG_1.Q OR R_TRIG_4.Q); // RS
Motor_Stop(Execute := Stopp.Q1, Deceleration := 100, Axis := Drive1); // MC_Stop
Motor_Stopped := Motor_Stop.Done;

// NETWORK 3
R_TRIG_0(CLK := Mode_Selected); // R_TRIG
TON_0(IN := NOT Mode_Selected OR NOT SCC_Motor_ON AND autoMode, PT := T#0.02s); // TON
Power_On_1(SET := R_TRIG_0.Q OR SCC_Motor_ON AND autoMode, RESET1 := TON_0.Q OR stopBtn AND Motor_Error); // RS
Motor_Power_On_0(Enable := Power_On_1.Q1, Axis := Drive1, Error => Motor_Error); // MC_Power
UDP_Send.PwrOn := Motor_Power_On_0.Status;
System_Ready := Motor_Power_On_0.Status;
SCC_On_Light := Motor_Power_On_0.Status;
Motor_Power_On := Motor_Power_On_0.Status;

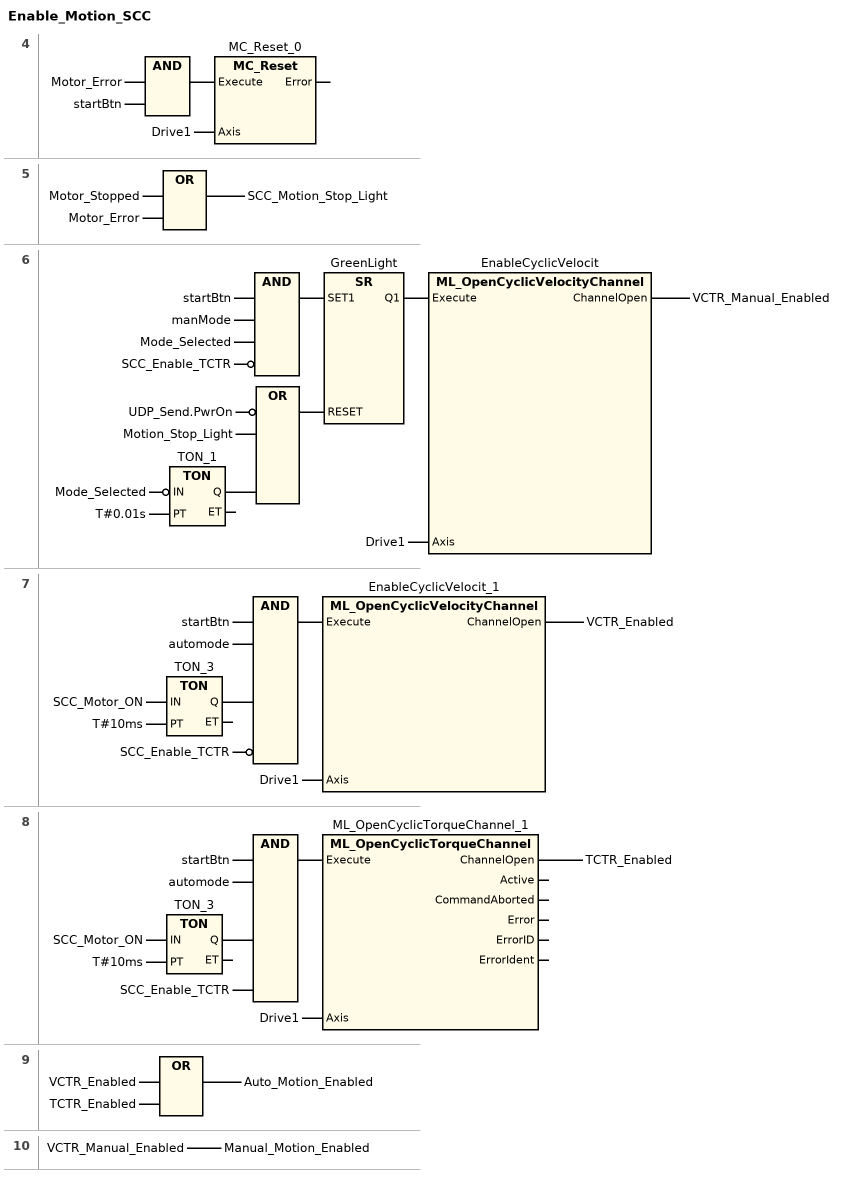
// NETWORK 4
MC_Reset_0(Execute := Motor_Error AND startBtn, Axis := Drive1); // MC_Reset

// NETWORK 5
SCC_Motion_Stop_Light := Motor_Stopped OR Motor_Error;

// NETWORK 6
TON_1(IN := NOT Mode_Selected, PT := T#0.01s); // TON
GreenLight(SET1 := startBtn AND manMode AND Mode_Selected AND NOT SCC_Enable_TCTR, RESET := NOT UDP_Send.PwrOn OR Motion_Stop_Light OR TON_1.Q); // SR
EnableCyclicVelocit(Execute := GreenLight.Q1, Axis := Drive1); // ML_OpenCyclicVelocityChannel
VCTR_Manual_Enabled := EnableCyclicVelocit.ChannelOpen;

// NETWORK 7
TON_3(IN := SCC_Motor_ON, PT := T#10ms); // TON
EnableCyclicVelocit_1(Execute := startBtn AND automode AND TON_3.Q AND NOT SCC_Enable_TCTR, Axis := Drive1); // ML_OpenCyclicVelocityChannel
VCTR_Enabled := EnableCyclicVelocit_1.ChannelOpen;

// NETWORK 8
TON_3(IN := SCC_Motor_ON, PT := T#10ms); // TON
ML_OpenCyclicTorqueChannel_1(Execute := startBtn AND automode AND TON_3.Q AND SCC_Enable_TCTR, Axis := Drive1); // ML_OpenCyclicTorqueChannel
TCTR_Enabled := ML_OpenCyclicTorqueChannel_1.ChannelOpen;

// NETWORK 9
Auto_Motion_Enabled := VCTR_Enabled OR TCTR_Enabled;

// NETWORK 10
Manual_Motion_Enabled := VCTR_Manual_Enabled;

END_FUNCTION_BLOCK

// IndraMotionMlc1/Application/Real_Time_Counter
FUNCTION_BLOCK Real_Time_Counter
VAR_INPUT
	Enable: BOOL;
	Start_Counter: BOOL;
END_VAR
VAR_OUTPUT
	Real_Time: LREAL;
END_VAR
VAR
	timereset: REAL;
END_VAR
VAR // added by the converter: edge detectors and wires of the graphical bodies
    _w1 : BOOL;
END_VAR

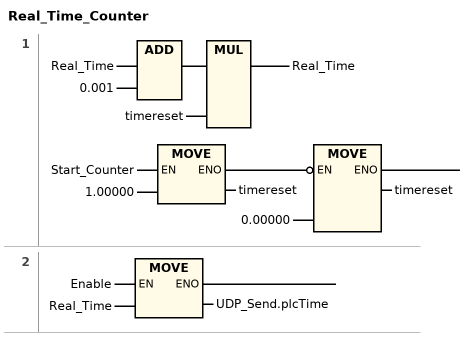
// NETWORK 1
Real_Time := (Real_Time + 0.001) * timereset;
_w1 := Start_Counter;
IF _w1 THEN timereset := 1.00000; END_IF
IF NOT _w1 THEN timereset := 0.00000; END_IF

// NETWORK 2
IF Enable THEN UDP_Send.plcTime := Real_Time; END_IF

END_FUNCTION_BLOCK

// IndraMotionMlc1/Application/LoadHolding_Control
FUNCTION_BLOCK LoadHolding_Control
VAR_INPUT
Enable: BOOL; 	
LH_auto_enable: BOOL;	
Force_Open: BOOL;
END_VAR
VAR_OUTPUT
LH_Valve_Open: BOOL;
END_VAR
VAR
LHactive: SR;
valveOn: BOOL;
END_VAR
VAR // added by the converter: edge detectors and wires of the graphical bodies
    _w1 : BOOL;
END_VAR

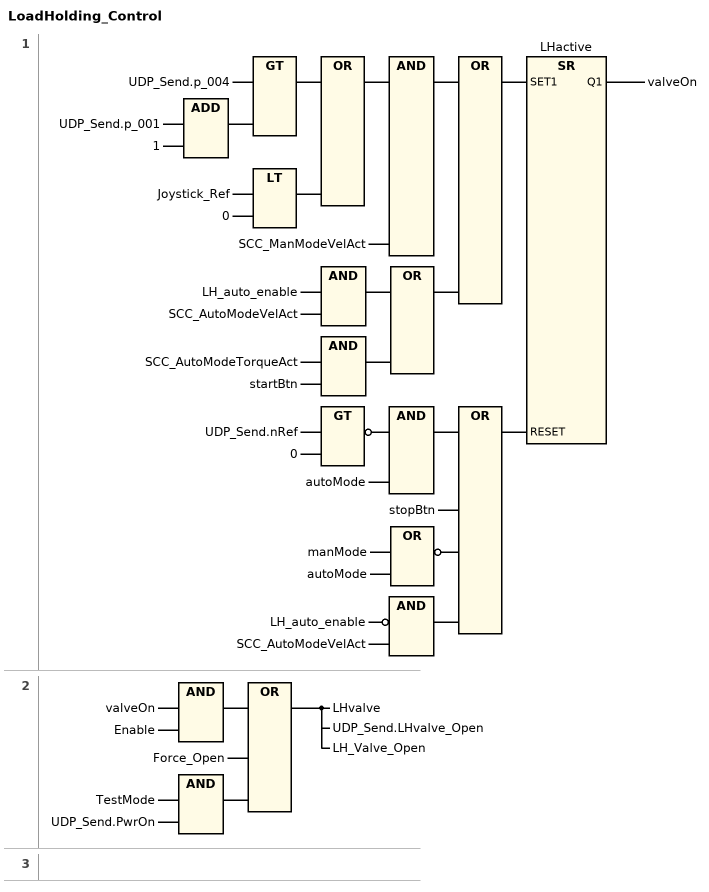
// NETWORK 1
LHactive(SET1 := (UDP_Send.p_004 > UDP_Send.p_001 + 1 OR Joystick_Ref < 0) AND SCC_ManModeVelAct OR (LH_auto_enable AND SCC_AutoModeVelAct OR SCC_AutoModeTorqueAct AND startBtn), RESET := NOT (UDP_Send.nRef > 0) AND autoMode OR stopBtn OR NOT (manMode OR autoMode) OR NOT LH_auto_enable AND SCC_AutoModeVelAct); // SR
valveOn := LHactive.Q1;

// NETWORK 2
_w1 := valveOn AND Enable OR Force_Open OR TestMode AND UDP_Send.PwrOn;
LHvalve := _w1;
UDP_Send.LHvalve_Open := _w1;
LH_Valve_Open := _w1;

// NETWORK 3

END_FUNCTION_BLOCK

// IndraMotionMlc1/Application/JoyStick_SCC
FUNCTION_BLOCK JoyStick_SCC
VAR_INPUT
	Enable: BOOL; 
	Max_Motor_Speed: REAL; 
END_VAR
VAR_OUTPUT
	JoyY_Ref: REAL;
END_VAR
VAR
END_VAR
VAR // added by the converter: edge detectors and wires of the graphical bodies
    _w1 : INT;
END_VAR

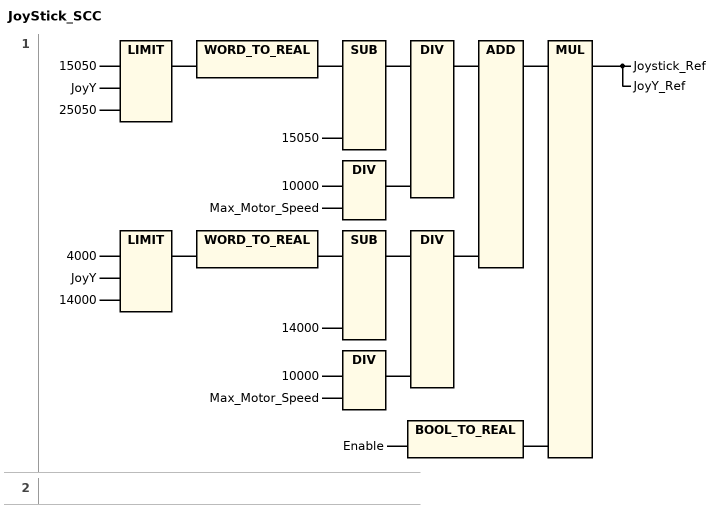
// NETWORK 1
_w1 := ((WORD_TO_REAL(LIMIT(15050, JoyY, 25050)) - 15050) / (10000 / Max_Motor_Speed) + (WORD_TO_REAL(LIMIT(4000, JoyY, 14000)) - 14000) / (10000 / Max_Motor_Speed)) * BOOL_TO_REAL(Enable);
Joystick_Ref := _w1;
JoyY_Ref := _w1;

// NETWORK 2

END_FUNCTION_BLOCK

// IndraMotionMlc1/Application/SCC_Controller
FUNCTION_BLOCK SCC_Controller
VAR_INPUT
	 Enable: BOOL;
END_VAR
VAR_OUTPUT
	 n_Ref: LREAL;
	 Position_Error: LREAL;
	 LHenable: BOOL;
END_VAR
VAR
	 VCC_Joystick_vel_ref_1: VCC_Joystick_vel_ref;
	 Vel_Ref_Joystick: LREAL;
	 AutoPLCtime_start: LREAL;
	 SPtime: LREAL;
	 SPtimereset: LREAL; 
	 S_shape_Profile_1: S_shape_Profile;
	 Ramp_Profile_0: Ramp_Profile;
	 CC_PI_FF_AD_0: CC_PI_FF_AD;
	 ActiveLH: BOOL;
	 k_P: LREAL;
	 Vel_Ref_Manual: LREAL;
	 Pos_Ref_Gen: LREAL;
	 Vel_Ref: LREAL;
     Pos_Ref: LREAL;
	 Ramp_Pos_Ref_Gen: LREAL;
	 Ramp_Vel_Ref_Gen: LREAL;
	 S_shape_Pos_Ref_Gen: LREAL;
	 S_shape_Vel_Ref_Gen: LREAL;
	 SP_Gen_Vel_Ref: LREAL;
     T_Ramp: LREAL;
	 T_S_shape: LREAL;
	SCC_Controller_FF_PI_AD_0: SCC_Controller_FF_PI_AD;
	LH_Passive_On: BOOL;
	Step_Damiano_0: Step_Damiano;
	StepTestTime: LREAL;
	SCC_Ramp_Test_0: SCC_Ramp_Test;
	SCC_HPPF_0: SCC_HPPF;
	uPF: LREAL;
	uEM_Ramp: LREAL;
	uEM: LREAL;
	uFF: LREAL;
	vRef: LREAL;
	TON_0: TON;
	SCC_LPPF_0: SCC_LPPF;
	SCC_DPF_0: SCC_DPF;
	uHPPF: LREAL;
	uLPPF: LREAL;
	uDPF: LREAL;
	SCC_Controller_PFB_0: SCC_Controller_PFB;
	SCC_Controller_VFF_0: SCC_Controller_VFF;
	uFB: LREAL;
	SCC_PFB_Controller_PID_0: SCC_PFB_Controller_PID;
	SCC_PFB_Controller_PID2_0: SCC_PFB_Controller_PID2;
	D_On: BOOL;
	n1: LREAL;
	n2: LREAL;
	d1: LREAL;
	d2: LREAL;
	d3: LREAL;
	SinuousCurve_Test_0: SinuousCurve_Test;
	SCC_SinProfile_0: SCC_SinProfile;
	Sin_Vel_Ref_Gen: LREAL;
	Sin_Pos_Ref_Gen: LREAL;
	CascadedControllerFilter_0: CascadedControllerFilter;
	CCF_ON: BOOL;
	CCF_N2: LREAL;
	CCF_N3: LREAL;
	CCF_D2: LREAL;
	CCF_D3: LREAL;
	uFB_Org: LREAL;
	uFB_CCF: LREAL;
	Motion_Enable_Timer: BOOL;
	LHV_Controller_0: LHV_Controller;
	uLHC: LREAL;
	LHV_Enabler_0: LHV_Enabler;
	LHV_error: LREAL;
	SM_ON: BOOL;
	uFF_uLHC: LREAL;
	SR_0: SR;
	TON_1: TON;
	TON_2: TON;
	uLHC1: LREAL;
	Pressure_Feed_Forward_0: Pressure_Feed_Forward;
	uPFF: LREAL;
	TON_3: TON;
	LHenable_ref: BOOL;
	SR_1: SR;
	PFF_tHold: BOOL;
	TON_4: TON;
	F_TRIG_0: F_TRIG;
	R_TRIG_0: R_TRIG;
	PFF_tHold_reset: BOOL;
	SR_2: SR;
	TON_5: TON;
	PFF_Active: BOOL;
	test22: BOOL;
	TON_6: TON;
	PFF_tHold_reset2: BOOL;
	R_TRIG_1: R_TRIG;
	PFF_tHold2: BOOL;
	test21: BOOL;
	uFB_uLHC: LREAL;
	SCC_Controller_PFB1_0: SCC_Controller_PFB1;
	uFB_uFF: LREAL;
	SCC_Vel_AD_0: SCC_Vel_AD;
	u_vel_AD: LREAL;
	SCC_VFF_0: SCC_VFF;
	k_I: LREAL;
	SCC_HPPF1_0: SCC_HPPF1;
	reset_PFF_delay: BOOL;
	uFF_uFB_uLHC: LREAL;
	uPF_1: LREAL;
	SR_3: SR;
	PF_ON: BOOL;
	F_TRIG_1: F_TRIG;
	SR_4: SR;
	TON_7: TON;
	LH_HOld: BOOL;
	R_TRIG_2: R_TRIG;
	R_TRIG_3: R_TRIG;
	FB_ON: BOOL;
	LHV_Controller2_0: LHV_Controller2;
	TON_8: TON;
	uPFF_ON: BOOL;
	TON_9: TON;
	SCC_LHC_On2: BOOL;
	SCC_LHC_On3: BOOL;
	TON_10: TON;
	TON_11: TON;
	TON_12: TON;
	Delay_Vel_0: Delay_Vel;
	Delay_Pos_0: Delay_Pos;
	VCC_Pos_Step_0: VCC_Pos_Step;
	Step_Pos_Ref: LREAL;
	TON_13: TON;
	SR_5: SR;
	R_TRIG_4: R_TRIG;
	F_TRIG_2: F_TRIG;
	R_TRIG_5: R_TRIG;
	
	FB_CTR_Test: BOOL := 1;
	SCC_AD_Iq_0: SCC_AD_Iq;
	uAD_Iq: LREAL;
	SCC_Acceleration_Feedback_0: SCC_Acceleration_Feedback;
	uAF: LREAL;
END_VAR
VAR // added by the converter: edge detectors and wires of the graphical bodies
    _w1 : INT;
    _w2, _w3, _w4, _w5, _w6, _w7, _w8, _w9, _w10, _w11, _w12, _w13, _w14, _w15, _w16, _w17 : BOOL;
END_VAR

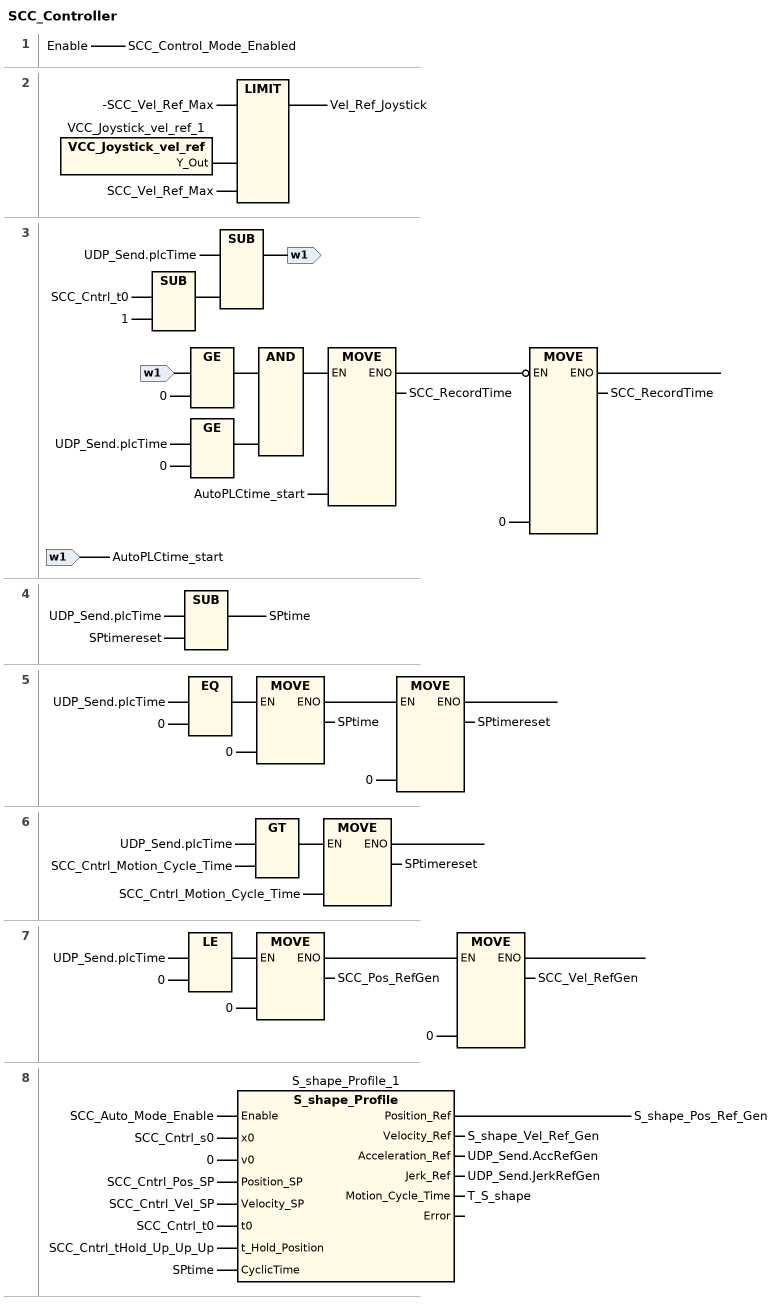
// NETWORK 1
SCC_Control_Mode_Enabled := Enable;

// NETWORK 2
VCC_Joystick_vel_ref_1(); // VCC_Joystick_vel_ref
Vel_Ref_Joystick := LIMIT(-SCC_Vel_Ref_Max, VCC_Joystick_vel_ref_1.Y_Out, SCC_Vel_Ref_Max);

// NETWORK 3
_w1 := UDP_Send.plcTime - (SCC_Cntrl_t0 - 1);
IF _w1 >= 0 AND UDP_Send.plcTime >= 0 THEN SCC_RecordTime := AutoPLCtime_start; END_IF
IF NOT (_w1 >= 0 AND UDP_Send.plcTime >= 0) THEN SCC_RecordTime := 0; END_IF
AutoPLCtime_start := _w1;

// NETWORK 4
SPtime := UDP_Send.plcTime - SPtimereset;

// NETWORK 5
_w2 := UDP_Send.plcTime = 0;
IF _w2 THEN SPtime := 0; END_IF
IF _w2 THEN SPtimereset := 0; END_IF

// NETWORK 6
IF UDP_Send.plcTime > SCC_Cntrl_Motion_Cycle_Time THEN SPtimereset := SCC_Cntrl_Motion_Cycle_Time; END_IF

// NETWORK 7
_w3 := UDP_Send.plcTime <= 0;
IF _w3 THEN SCC_Pos_RefGen := 0; END_IF
IF _w3 THEN SCC_Vel_RefGen := 0; END_IF

// NETWORK 8
S_shape_Profile_1(
    Enable := SCC_Auto_Mode_Enable,
    x0 := SCC_Cntrl_s0,
    v0 := 0,
    Position_SP := SCC_Cntrl_Pos_SP,
    Velocity_SP := SCC_Cntrl_Vel_SP,
    t0 := SCC_Cntrl_t0,
    t_Hold_Position := SCC_Cntrl_tHold_Up_Up_Up,
    CyclicTime := SPtime,
    Velocity_Ref => S_shape_Vel_Ref_Gen,
    Acceleration_Ref => UDP_Send.AccRefGen,
    Jerk_Ref => UDP_Send.JerkRefGen,
    Motion_Cycle_Time => T_S_shape); // S_shape_Profile
S_shape_Pos_Ref_Gen := S_shape_Profile_1.Position_Ref;

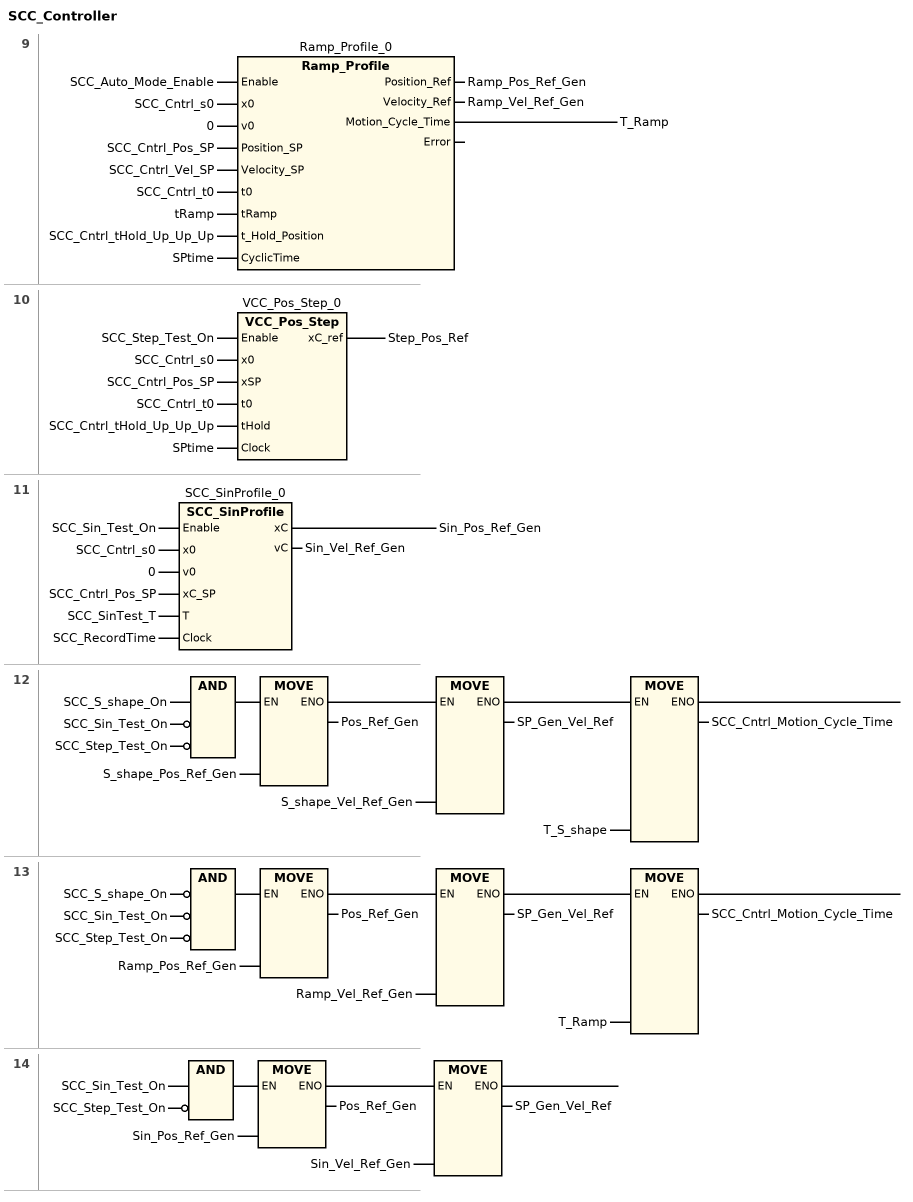
// NETWORK 9
Ramp_Profile_0(
    Enable := SCC_Auto_Mode_Enable,
    x0 := SCC_Cntrl_s0,
    v0 := 0,
    Position_SP := SCC_Cntrl_Pos_SP,
    Velocity_SP := SCC_Cntrl_Vel_SP,
    t0 := SCC_Cntrl_t0,
    tRamp := tRamp,
    t_Hold_Position := SCC_Cntrl_tHold_Up_Up_Up,
    CyclicTime := SPtime,
    Position_Ref => Ramp_Pos_Ref_Gen,
    Velocity_Ref => Ramp_Vel_Ref_Gen); // Ramp_Profile
T_Ramp := Ramp_Profile_0.Motion_Cycle_Time;

// NETWORK 10
VCC_Pos_Step_0(
    Enable := SCC_Step_Test_On,
    x0 := SCC_Cntrl_s0,
    xSP := SCC_Cntrl_Pos_SP,
    t0 := SCC_Cntrl_t0,
    tHold := SCC_Cntrl_tHold_Up_Up_Up,
    Clock := SPtime); // VCC_Pos_Step
Step_Pos_Ref := VCC_Pos_Step_0.xC_ref;

// NETWORK 11
SCC_SinProfile_0(
    Enable := SCC_Sin_Test_On,
    x0 := SCC_Cntrl_s0,
    v0 := 0,
    xC_SP := SCC_Cntrl_Pos_SP,
    T := SCC_SinTest_T,
    Clock := SCC_RecordTime,
    vC => Sin_Vel_Ref_Gen); // SCC_SinProfile
Sin_Pos_Ref_Gen := SCC_SinProfile_0.xC;

// NETWORK 12
_w4 := SCC_S_shape_On AND NOT SCC_Sin_Test_On AND NOT SCC_Step_Test_On;
IF _w4 THEN Pos_Ref_Gen := S_shape_Pos_Ref_Gen; END_IF
IF _w4 THEN SP_Gen_Vel_Ref := S_shape_Vel_Ref_Gen; END_IF
IF _w4 THEN SCC_Cntrl_Motion_Cycle_Time := T_S_shape; END_IF

// NETWORK 13
_w5 := NOT SCC_S_shape_On AND NOT SCC_Sin_Test_On AND NOT SCC_Step_Test_On;
IF _w5 THEN Pos_Ref_Gen := Ramp_Pos_Ref_Gen; END_IF
IF _w5 THEN SP_Gen_Vel_Ref := Ramp_Vel_Ref_Gen; END_IF
IF _w5 THEN SCC_Cntrl_Motion_Cycle_Time := T_Ramp; END_IF

// NETWORK 14
_w6 := SCC_Sin_Test_On AND NOT SCC_Step_Test_On;
IF _w6 THEN Pos_Ref_Gen := Sin_Pos_Ref_Gen; END_IF
IF _w6 THEN SP_Gen_Vel_Ref := Sin_Vel_Ref_Gen; END_IF

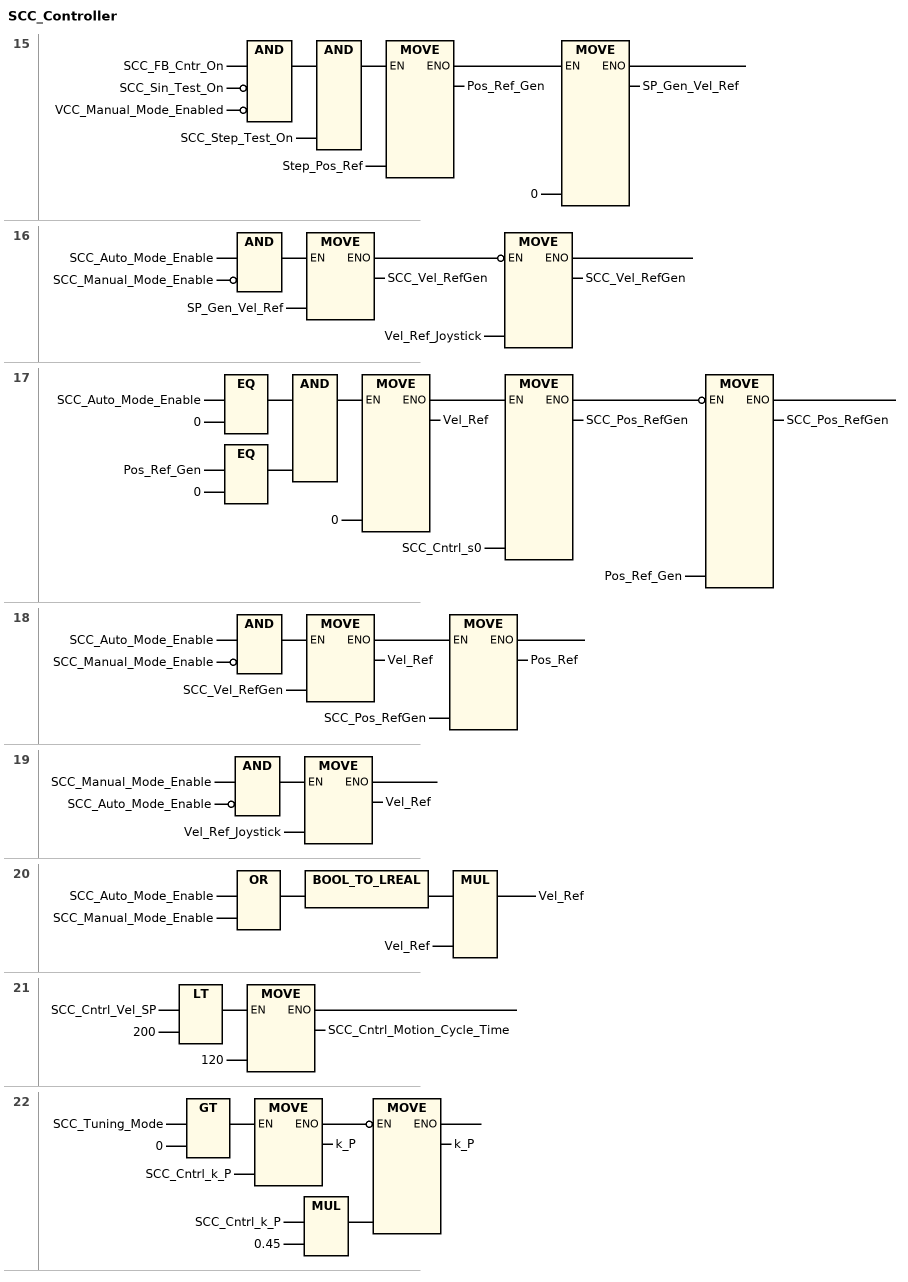
// NETWORK 15
_w7 := (SCC_FB_Cntr_On AND NOT SCC_Sin_Test_On AND NOT VCC_Manual_Mode_Enabled) AND SCC_Step_Test_On;
IF _w7 THEN Pos_Ref_Gen := Step_Pos_Ref; END_IF
IF _w7 THEN SP_Gen_Vel_Ref := 0; END_IF

// NETWORK 16
_w8 := SCC_Auto_Mode_Enable AND NOT SCC_Manual_Mode_Enable;
IF _w8 THEN SCC_Vel_RefGen := SP_Gen_Vel_Ref; END_IF
IF NOT _w8 THEN SCC_Vel_RefGen := Vel_Ref_Joystick; END_IF

// NETWORK 17
_w9 := SCC_Auto_Mode_Enable = 0 AND Pos_Ref_Gen = 0;
IF _w9 THEN Vel_Ref := 0; END_IF
IF _w9 THEN SCC_Pos_RefGen := SCC_Cntrl_s0; END_IF
IF NOT _w9 THEN SCC_Pos_RefGen := Pos_Ref_Gen; END_IF

// NETWORK 18
_w10 := SCC_Auto_Mode_Enable AND NOT SCC_Manual_Mode_Enable;
IF _w10 THEN Vel_Ref := SCC_Vel_RefGen; END_IF
IF _w10 THEN Pos_Ref := SCC_Pos_RefGen; END_IF

// NETWORK 19
IF SCC_Manual_Mode_Enable AND NOT SCC_Auto_Mode_Enable THEN Vel_Ref := Vel_Ref_Joystick; END_IF

// NETWORK 20
Vel_Ref := BOOL_TO_LREAL(SCC_Auto_Mode_Enable OR SCC_Manual_Mode_Enable) * Vel_Ref;

// NETWORK 21
IF SCC_Cntrl_Vel_SP < 200 THEN SCC_Cntrl_Motion_Cycle_Time := 120; END_IF

// NETWORK 22
_w11 := SCC_Tuning_Mode > 0;
IF _w11 THEN k_P := SCC_Cntrl_k_P; END_IF
IF NOT _w11 THEN k_P := SCC_Cntrl_k_P * 0.45; END_IF

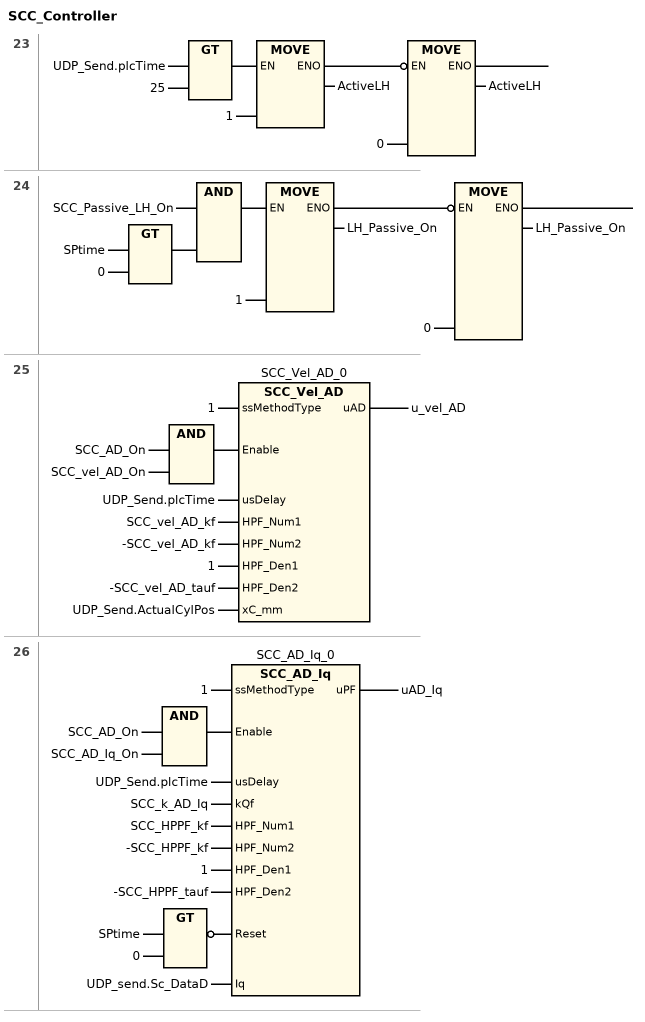
// NETWORK 23
_w12 := UDP_Send.plcTime > 25;
IF _w12 THEN ActiveLH := 1; END_IF
IF NOT _w12 THEN ActiveLH := 0; END_IF

// NETWORK 24
_w13 := SCC_Passive_LH_On AND SPtime > 0;
IF _w13 THEN LH_Passive_On := 1; END_IF
IF NOT _w13 THEN LH_Passive_On := 0; END_IF

// NETWORK 25
SCC_Vel_AD_0(
    ssMethodType := 1,
    Enable := SCC_AD_On AND SCC_vel_AD_On,
    usDelay := UDP_Send.plcTime,
    HPF_Num1 := SCC_vel_AD_kf,
    HPF_Num2 := -SCC_vel_AD_kf,
    HPF_Den1 := 1,
    HPF_Den2 := -SCC_vel_AD_tauf,
    xC_mm := UDP_Send.ActualCylPos); // SCC_Vel_AD
u_vel_AD := SCC_Vel_AD_0.uAD;

// NETWORK 26
SCC_AD_Iq_0(
    ssMethodType := 1,
    Enable := SCC_AD_On AND SCC_AD_Iq_On,
    usDelay := UDP_Send.plcTime,
    kQf := SCC_k_AD_Iq,
    HPF_Num1 := SCC_HPPF_kf,
    HPF_Num2 := -SCC_HPPF_kf,
    HPF_Den1 := 1,
    HPF_Den2 := -SCC_HPPF_tauf,
    Reset := NOT (SPtime > 0),
    Iq := UDP_send.Sc_DataD); // SCC_AD_Iq
uAD_Iq := SCC_AD_Iq_0.uPF;

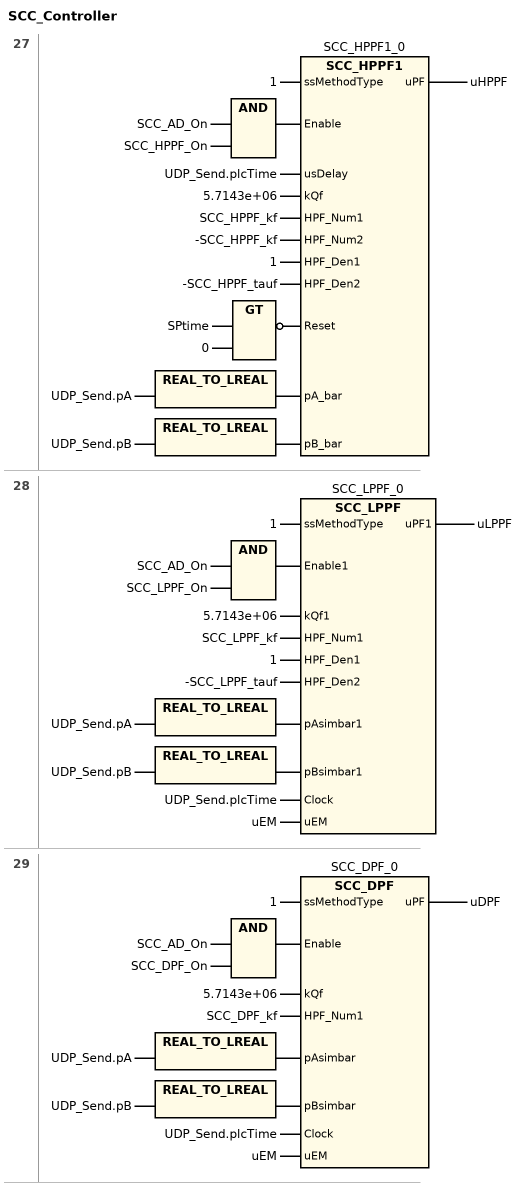
// NETWORK 27
SCC_HPPF1_0(
    ssMethodType := 1,
    Enable := SCC_AD_On AND SCC_HPPF_On,
    usDelay := UDP_Send.plcTime,
    kQf := 5.7143e+06,
    HPF_Num1 := SCC_HPPF_kf,
    HPF_Num2 := -SCC_HPPF_kf,
    HPF_Den1 := 1,
    HPF_Den2 := -SCC_HPPF_tauf,
    Reset := NOT (SPtime > 0),
    pA_bar := REAL_TO_LREAL(UDP_Send.pA),
    pB_bar := REAL_TO_LREAL(UDP_Send.pB)); // SCC_HPPF1
uHPPF := SCC_HPPF1_0.uPF;

// NETWORK 28
SCC_LPPF_0(
    ssMethodType := 1,
    Enable1 := SCC_AD_On AND SCC_LPPF_On,
    kQf1 := 5.7143e+06,
    HPF_Num1 := SCC_LPPF_kf,
    HPF_Den1 := 1,
    HPF_Den2 := -SCC_LPPF_tauf,
    pAsimbar1 := REAL_TO_LREAL(UDP_Send.pA),
    pBsimbar1 := REAL_TO_LREAL(UDP_Send.pB),
    Clock := UDP_Send.plcTime,
    uEM := uEM); // SCC_LPPF
uLPPF := SCC_LPPF_0.uPF1;

// NETWORK 29
SCC_DPF_0(
    ssMethodType := 1,
    Enable := SCC_AD_On AND SCC_DPF_On,
    kQf := 5.7143e+06,
    HPF_Num1 := SCC_DPF_kf,
    pAsimbar := REAL_TO_LREAL(UDP_Send.pA),
    pBsimbar := REAL_TO_LREAL(UDP_Send.pB),
    Clock := UDP_Send.plcTime,
    uEM := uEM); // SCC_DPF
uDPF := SCC_DPF_0.uPF;

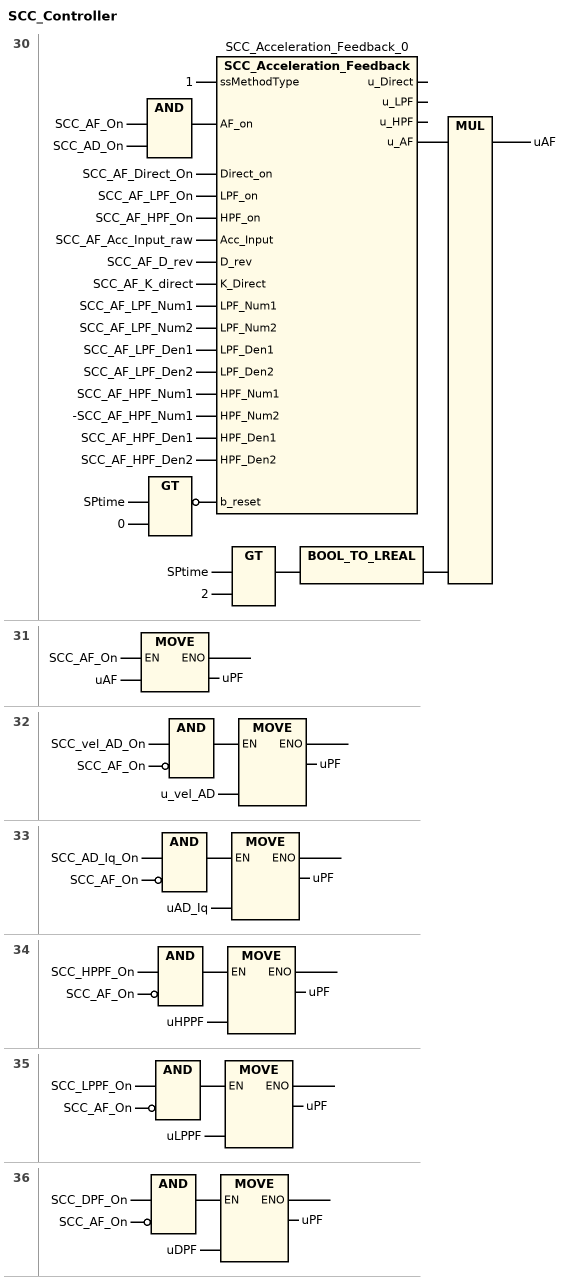
// NETWORK 30
SCC_Acceleration_Feedback_0(
    ssMethodType := 1,
    AF_on := SCC_AF_On AND SCC_AD_On,
    Direct_on := SCC_AF_Direct_On,
    LPF_on := SCC_AF_LPF_On,
    HPF_on := SCC_AF_HPF_On,
    Acc_Input := SCC_AF_Acc_Input_raw,
    D_rev := SCC_AF_D_rev,
    K_Direct := SCC_AF_K_direct,
    LPF_Num1 := SCC_AF_LPF_Num1,
    LPF_Num2 := SCC_AF_LPF_Num2,
    LPF_Den1 := SCC_AF_LPF_Den1,
    LPF_Den2 := SCC_AF_LPF_Den2,
    HPF_Num1 := SCC_AF_HPF_Num1,
    HPF_Num2 := -SCC_AF_HPF_Num1,
    HPF_Den1 := SCC_AF_HPF_Den1,
    HPF_Den2 := SCC_AF_HPF_Den2,
    b_reset := NOT (SPtime > 0)); // SCC_Acceleration_Feedback
uAF := SCC_Acceleration_Feedback_0.u_AF * BOOL_TO_LREAL(SPtime > 2);

// NETWORK 31
IF SCC_AF_On THEN uPF := uAF; END_IF

// NETWORK 32
IF SCC_vel_AD_On AND NOT SCC_AF_On THEN uPF := u_vel_AD; END_IF

// NETWORK 33
IF SCC_AD_Iq_On AND NOT SCC_AF_On THEN uPF := uAD_Iq; END_IF

// NETWORK 34
IF SCC_HPPF_On AND NOT SCC_AF_On THEN uPF := uHPPF; END_IF

// NETWORK 35
IF SCC_LPPF_On AND NOT SCC_AF_On THEN uPF := uLPPF; END_IF

// NETWORK 36
IF SCC_DPF_On AND NOT SCC_AF_On THEN uPF := uDPF; END_IF

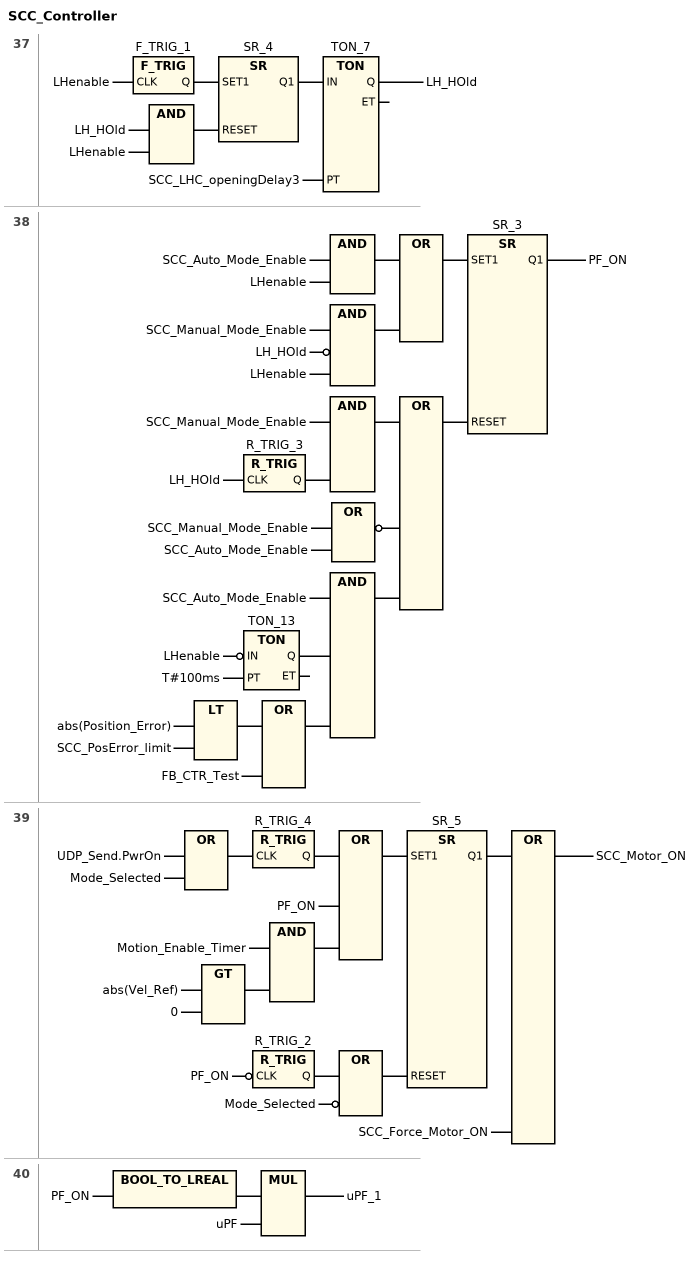
// NETWORK 37
F_TRIG_1(CLK := LHenable); // F_TRIG
SR_4(SET1 := F_TRIG_1.Q, RESET := LH_HOld AND LHenable); // SR
TON_7(IN := SR_4.Q1, PT := SCC_LHC_openingDelay3); // TON
LH_HOld := TON_7.Q;

// NETWORK 38
R_TRIG_3(CLK := LH_HOld); // R_TRIG
TON_13(IN := NOT LHenable, PT := T#100ms); // TON
SR_3(SET1 := SCC_Auto_Mode_Enable AND LHenable OR SCC_Manual_Mode_Enable AND NOT LH_HOld AND LHenable, RESET := SCC_Manual_Mode_Enable AND R_TRIG_3.Q OR NOT (SCC_Manual_Mode_Enable OR SCC_Auto_Mode_Enable) OR SCC_Auto_Mode_Enable AND TON_13.Q AND ((abs(Position_Error)) < SCC_PosError_limit OR FB_CTR_Test)); // SR
PF_ON := SR_3.Q1;

// NETWORK 39
R_TRIG_4(CLK := UDP_Send.PwrOn OR Mode_Selected); // R_TRIG
R_TRIG_2(CLK := NOT PF_ON); // R_TRIG
SR_5(SET1 := R_TRIG_4.Q OR PF_ON OR Motion_Enable_Timer AND (abs(Vel_Ref)) > 0, RESET := R_TRIG_2.Q OR NOT Mode_Selected); // SR
SCC_Motor_ON := SR_5.Q1 OR SCC_Force_Motor_ON;

// NETWORK 40
uPF_1 := BOOL_TO_LREAL(PF_ON) * uPF;

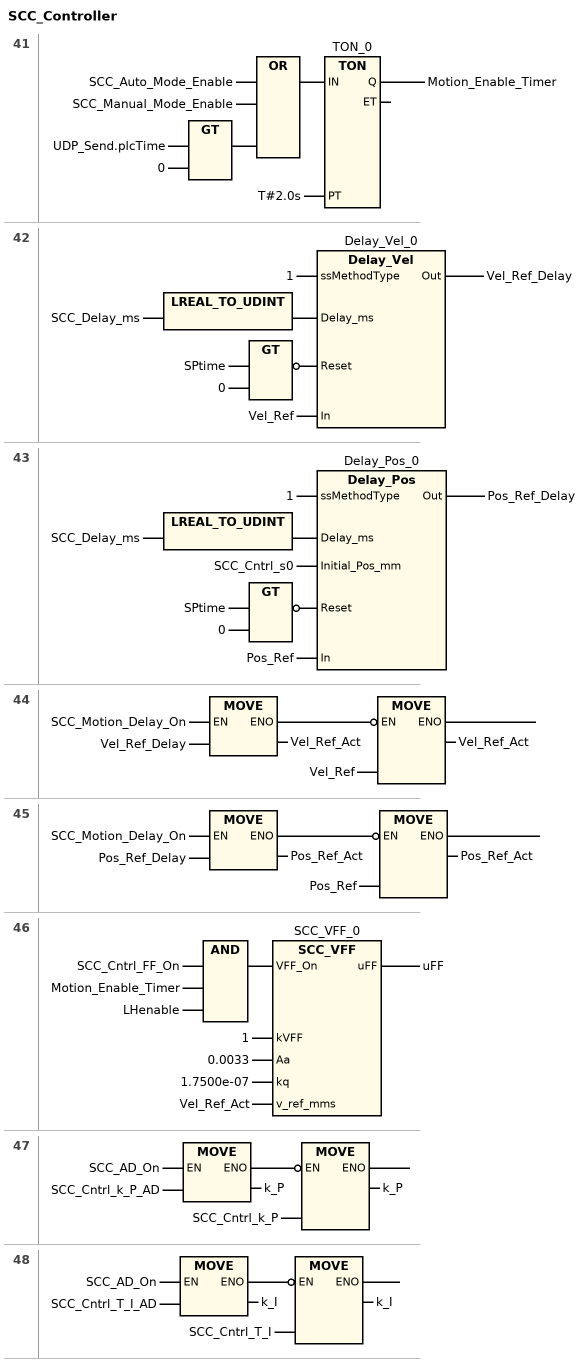
// NETWORK 41
TON_0(IN := SCC_Auto_Mode_Enable OR SCC_Manual_Mode_Enable OR UDP_Send.plcTime > 0, PT := T#2.0s); // TON
Motion_Enable_Timer := TON_0.Q;

// NETWORK 42
Delay_Vel_0(
    ssMethodType := 1,
    Delay_ms := LREAL_TO_UDINT(SCC_Delay_ms),
    Reset := NOT (SPtime > 0),
    In := Vel_Ref); // Delay_Vel
Vel_Ref_Delay := Delay_Vel_0.Out;

// NETWORK 43
Delay_Pos_0(
    ssMethodType := 1,
    Delay_ms := LREAL_TO_UDINT(SCC_Delay_ms),
    Initial_Pos_mm := SCC_Cntrl_s0,
    Reset := NOT (SPtime > 0),
    In := Pos_Ref); // Delay_Pos
Pos_Ref_Delay := Delay_Pos_0.Out;

// NETWORK 44
_w14 := SCC_Motion_Delay_On;
IF _w14 THEN Vel_Ref_Act := Vel_Ref_Delay; END_IF
IF NOT _w14 THEN Vel_Ref_Act := Vel_Ref; END_IF

// NETWORK 45
_w15 := SCC_Motion_Delay_On;
IF _w15 THEN Pos_Ref_Act := Pos_Ref_Delay; END_IF
IF NOT _w15 THEN Pos_Ref_Act := Pos_Ref; END_IF

// NETWORK 46
SCC_VFF_0(
    VFF_On := SCC_Cntrl_FF_On AND Motion_Enable_Timer AND LHenable,
    kVFF := 1,
    Aa := 0.0033,
    kq := 1.7500e-07,
    v_ref_mms := Vel_Ref_Act); // SCC_VFF
uFF := SCC_VFF_0.uFF;

// NETWORK 47
_w16 := SCC_AD_On;
IF _w16 THEN k_P := SCC_Cntrl_k_P_AD; END_IF
IF NOT _w16 THEN k_P := SCC_Cntrl_k_P; END_IF

// NETWORK 48
_w17 := SCC_AD_On;
IF _w17 THEN k_I := SCC_Cntrl_T_I_AD; END_IF
IF NOT _w17 THEN k_I := SCC_Cntrl_T_I; END_IF

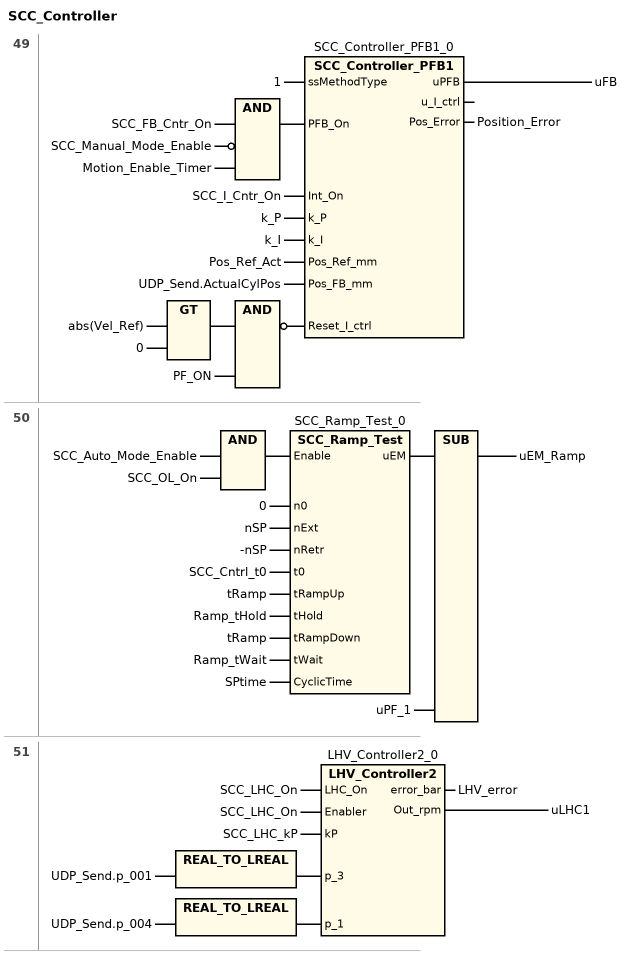
// NETWORK 49
SCC_Controller_PFB1_0(
    ssMethodType := 1,
    PFB_On := SCC_FB_Cntr_On AND NOT SCC_Manual_Mode_Enable AND Motion_Enable_Timer,
    Int_On := SCC_I_Cntr_On,
    k_P := k_P,
    k_I := k_I,
    Pos_Ref_mm := Pos_Ref_Act,
    Pos_FB_mm := UDP_Send.ActualCylPos,
    Reset_I_ctrl := NOT ((abs(Vel_Ref)) > 0 AND PF_ON),
    Pos_Error => Position_Error); // SCC_Controller_PFB1
uFB := SCC_Controller_PFB1_0.uPFB;

// NETWORK 50
SCC_Ramp_Test_0(
    Enable := SCC_Auto_Mode_Enable AND SCC_OL_On,
    n0 := 0,
    nExt := nSP,
    nRetr := -nSP,
    t0 := SCC_Cntrl_t0,
    tRampUp := tRamp,
    tHold := Ramp_tHold,
    tRampDown := tRamp,
    tWait := Ramp_tWait,
    CyclicTime := SPtime); // SCC_Ramp_Test
uEM_Ramp := SCC_Ramp_Test_0.uEM - uPF_1;

// NETWORK 51
LHV_Controller2_0(
    LHC_On := SCC_LHC_On,
    Enabler := SCC_LHC_On,
    kP := SCC_LHC_kP,
    p_3 := REAL_TO_LREAL(UDP_Send.p_001),
    p_1 := REAL_TO_LREAL(UDP_Send.p_004),
    error_bar => LHV_error); // LHV_Controller2
uLHC1 := LHV_Controller2_0.Out_rpm;

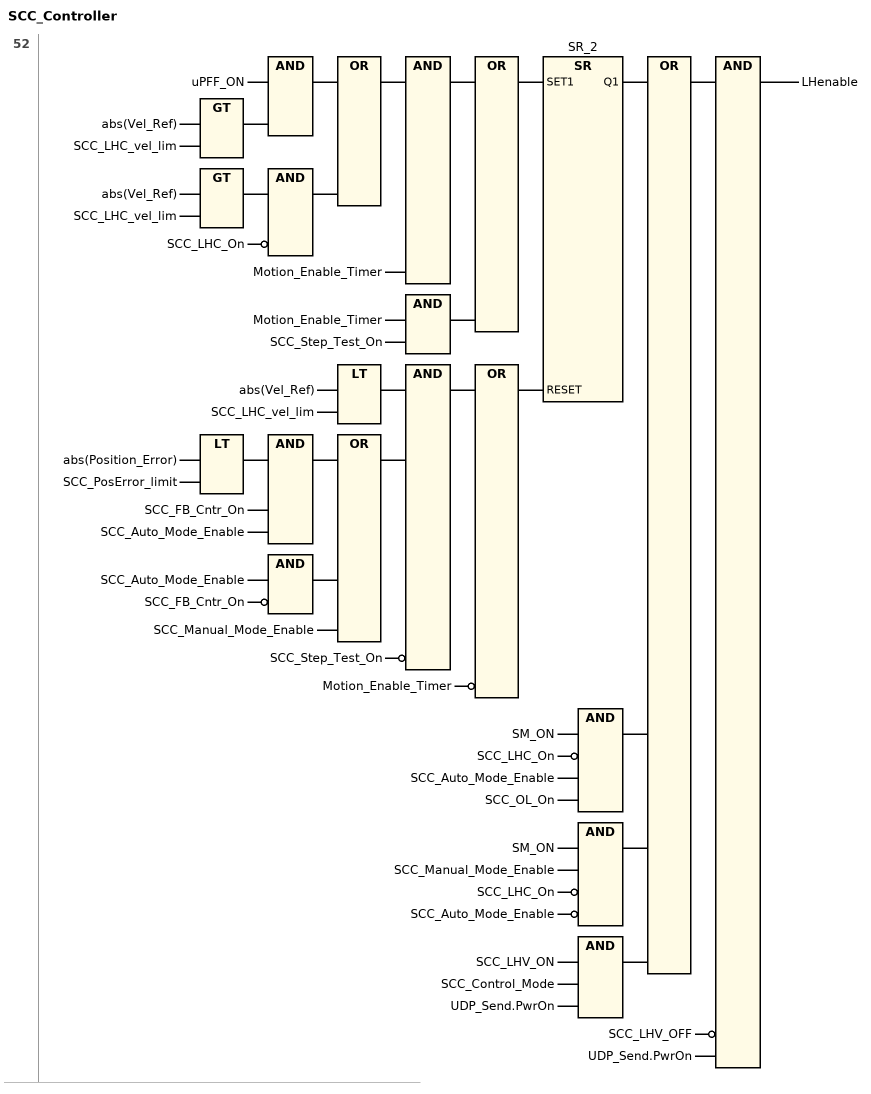
// NETWORK 52
SR_2(SET1 := (uPFF_ON AND (abs(Vel_Ref)) > SCC_LHC_vel_lim OR (abs(Vel_Ref)) > SCC_LHC_vel_lim AND NOT SCC_LHC_On) AND Motion_Enable_Timer OR Motion_Enable_Timer AND SCC_Step_Test_On, RESET := (abs(Vel_Ref)) < SCC_LHC_vel_lim AND ((abs(Position_Error)) < SCC_PosError_limit AND SCC_FB_Cntr_On AND SCC_Auto_Mode_Enable OR SCC_Auto_Mode_Enable AND NOT SCC_FB_Cntr_On OR SCC_Manual_Mode_Enable) AND NOT SCC_Step_Test_On OR NOT Motion_Enable_Timer); // SR
LHenable := (SR_2.Q1 OR SM_ON AND NOT SCC_LHC_On AND SCC_Auto_Mode_Enable AND SCC_OL_On OR SM_ON AND SCC_Manual_Mode_Enable AND NOT SCC_LHC_On AND NOT SCC_Auto_Mode_Enable OR SCC_LHV_ON AND SCC_Control_Mode AND UDP_Send.PwrOn) AND NOT SCC_LHV_OFF AND UDP_Send.PwrOn;

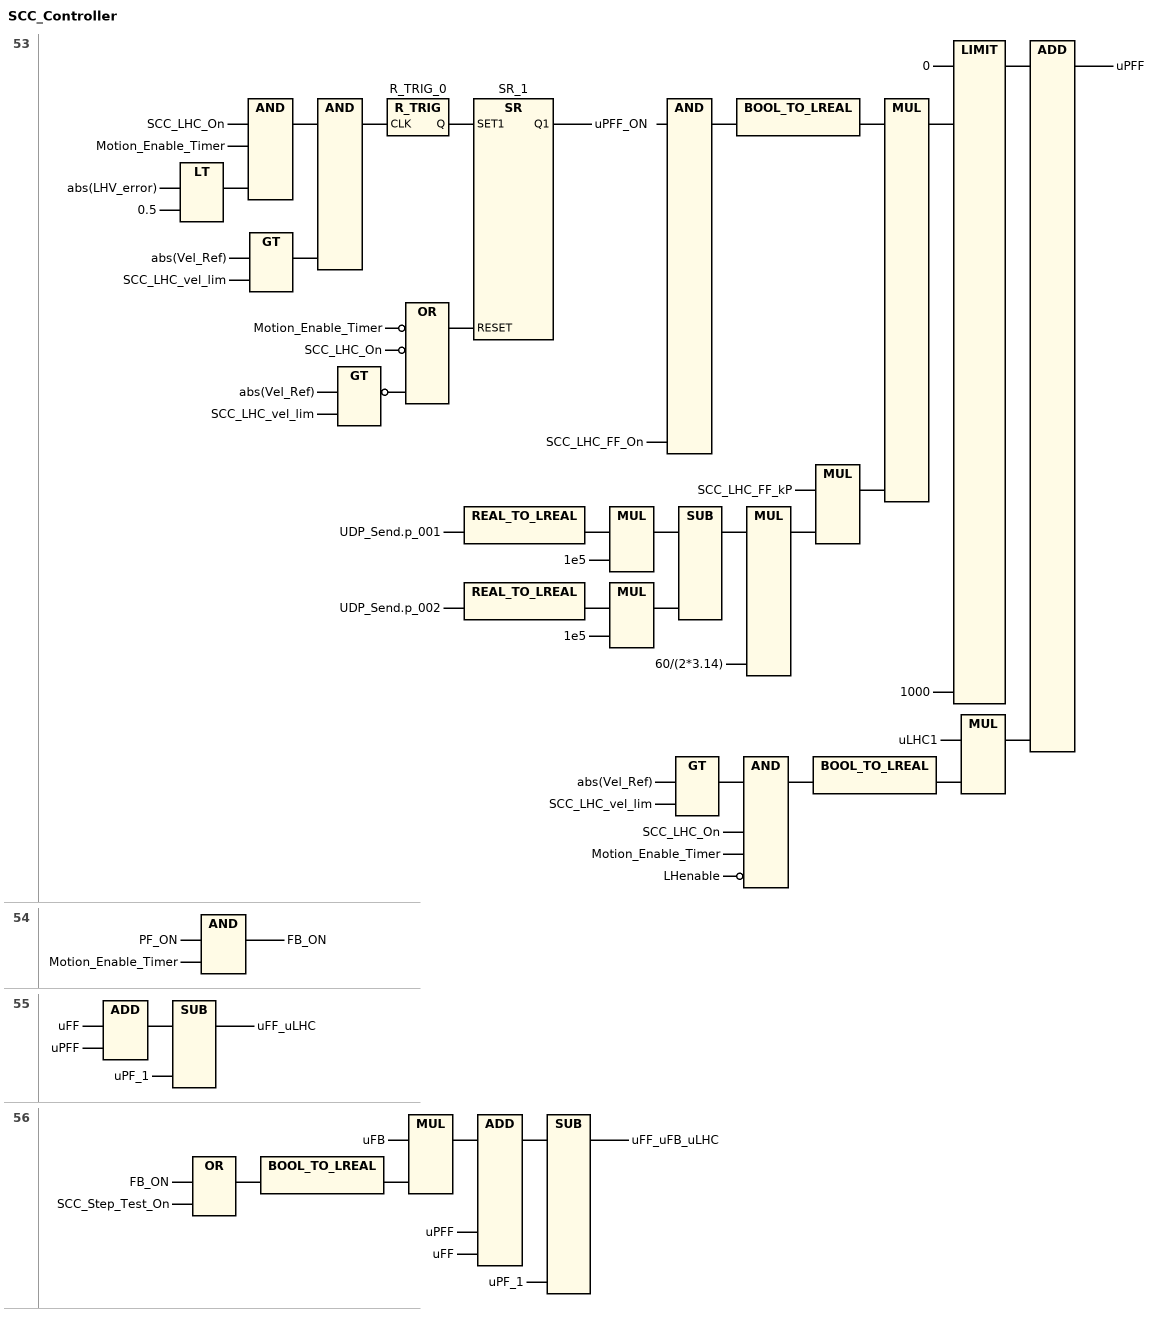
// NETWORK 53
R_TRIG_0(CLK := (SCC_LHC_On AND Motion_Enable_Timer AND (abs(LHV_error)) < 0.5) AND (abs(Vel_Ref)) > SCC_LHC_vel_lim); // R_TRIG
SR_1(SET1 := R_TRIG_0.Q, RESET := NOT Motion_Enable_Timer OR NOT SCC_LHC_On OR NOT ((abs(Vel_Ref)) > SCC_LHC_vel_lim)); // SR
uPFF_ON := SR_1.Q1;
uPFF := LIMIT(0, BOOL_TO_LREAL(SR_1.Q1 AND SCC_LHC_FF_On) * (SCC_LHC_FF_kP * ((REAL_TO_LREAL(UDP_Send.p_001) * 1e5 - REAL_TO_LREAL(UDP_Send.p_002) * 1e5) * (60/(2*3.14)))), 1000) + uLHC1 * BOOL_TO_LREAL((abs(Vel_Ref)) > SCC_LHC_vel_lim AND SCC_LHC_On AND Motion_Enable_Timer AND NOT LHenable);

// NETWORK 54
FB_ON := PF_ON AND Motion_Enable_Timer;

// NETWORK 55
uFF_uLHC := (uFF + uPFF) - uPF_1;

// NETWORK 56
uFF_uFB_uLHC := (uFB * BOOL_TO_LREAL(FB_ON OR SCC_Step_Test_On) + uPFF + uFF) - uPF_1;

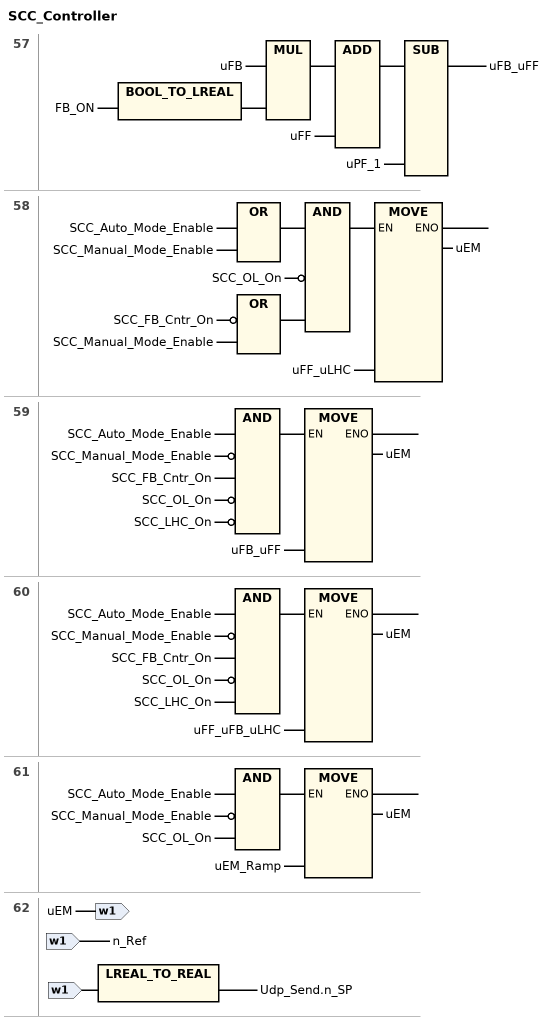
// NETWORK 57
uFB_uFF := (uFB * BOOL_TO_LREAL(FB_ON) + uFF) - uPF_1;

// NETWORK 58
IF (SCC_Auto_Mode_Enable OR SCC_Manual_Mode_Enable) AND NOT SCC_OL_On AND (NOT SCC_FB_Cntr_On OR SCC_Manual_Mode_Enable) THEN
    uEM := uFF_uLHC;
END_IF

// NETWORK 59
IF SCC_Auto_Mode_Enable AND NOT SCC_Manual_Mode_Enable AND SCC_FB_Cntr_On AND NOT SCC_OL_On AND NOT SCC_LHC_On THEN
    uEM := uFB_uFF;
END_IF

// NETWORK 60
IF SCC_Auto_Mode_Enable AND NOT SCC_Manual_Mode_Enable AND SCC_FB_Cntr_On AND NOT SCC_OL_On AND SCC_LHC_On THEN
    uEM := uFF_uFB_uLHC;
END_IF

// NETWORK 61
IF SCC_Auto_Mode_Enable AND NOT SCC_Manual_Mode_Enable AND SCC_OL_On THEN uEM := uEM_Ramp; END_IF

// NETWORK 62
n_Ref := uEM;
Udp_Send.n_SP := LREAL_TO_REAL(uEM);

END_FUNCTION_BLOCK

// IndraMotionMlc1/Application/VCC_Joystick_vel_ref
FUNCTION_BLOCK VCC_Joystick_vel_ref
VAR_INPUT
END_VAR
VAR_OUTPUT
	Y_Out: REAL;
END_VAR

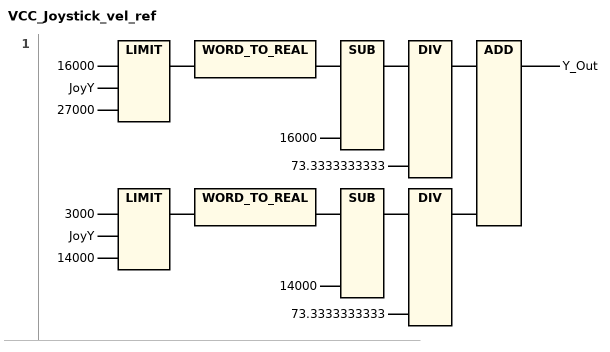
// NETWORK 1
Y_Out := (WORD_TO_REAL(LIMIT(16000, JoyY, 27000)) - 16000) / 73.3333333333 + (WORD_TO_REAL(LIMIT(3000, JoyY, 14000)) - 14000) / 73.3333333333;

END_FUNCTION_BLOCK

// IndraMotionMlc1/Application/S_shape_Profile
FUNCTION_BLOCK S_shape_Profile
VAR_INPUT
	Enable: BOOL;
	x0: LREAL;
	v0: LREAL;
	Position_SP: LREAL;
	Velocity_SP: LREAL;
	t0: LREAL;
	t_Hold_Position: LREAL;
	CyclicTime: LREAL;
END_VAR
VAR_OUTPUT
	Position_Ref: LREAL;
	Velocity_Ref: LREAL;
	Acceleration_Ref: LREAL;
	Jerk_Ref: LREAL;
	Motion_Cycle_Time: LREAL;
	Error: LREAL;
END_VAR
VAR
	Error_0: DINT;
	s_acc: LREAL;
	t1: LREAL;
	t2: LREAL;
	t3: LREAL;
	t4: LREAL;
	t6: LREAL;
	t7: LREAL;
	t8: LREAL;
	t9: LREAL;
	t10: LREAL;
	sh: LREAL;
	vh: LREAL;
	s3: LREAL;
	s4: LREAL;
	v4: LREAL;
	s7: LREAL;
	rtb_Saturation: LREAL;
	rtb_Saturation1: LREAL;
	t1_tmp: LREAL;
	temp1: BOOL;
END_VAR


(* Outputs for Atomic SubSystem: '<Root>/S_shape_Profile' *)
(* Saturate: '<S1>/Saturation' *)

IF Position_SP >= 500.0 THEN 
    rtb_Saturation := 500.0;
ELSIF Position_SP > 0.0 THEN 
    rtb_Saturation := Position_SP;
ELSE 
    rtb_Saturation := 0.0;
END_IF;

(* End of Saturate: '<S1>/Saturation' *)


(* Saturate: '<S1>/Saturation1' *)

IF Velocity_SP >= 150.0 THEN 
    rtb_Saturation1 := 150.0;
ELSIF Velocity_SP > -150.0 THEN 
    rtb_Saturation1 := Velocity_SP;
ELSE 
    rtb_Saturation1 := -150.0;
END_IF;

(* End of Saturate: '<S1>/Saturation1' *)


(* MATLAB Function: '<S1>/SP_Generator' *)
(* MATLAB Function 'S_shape_Profile/SP_Generator': '<S2>:1' *)
(* '<S2>:1:4' PositionSP = Desired_Position - s0; *)
(* '<S2>:1:6' a0 = 0; *)
(* '<S2>:1:7' j0 = 0; *)
(* '<S2>:1:8' AccelerationSP = VelocitySP; *)
(* '<S2>:1:10' vel=VelocitySP; *)
(* '<S2>:1:11' as=AccelerationSP; *)
(* Input velocity  *)
(* '<S2>:1:13' vs=vel; *)
(* [rad/s] *)
(* Delta velocity  *)
(* '<S2>:1:15' dv=(vs-v0); *)
(* [rad/s]      *)
(* Max Jerk Considerations *)
(* '<S2>:1:17' jm=as^2/dv; *)
sh := rtb_Saturation1 * rtb_Saturation1;
vh := rtb_Saturation1 - v0;
Jerk_Ref := sh / vh;
(* [rad/s^3]  *)
(* Constant Velocity periodes *)
(* '<S2>:1:19' s_acc=(vs^2-v0^2)/as; *)
s_acc := (sh - (v0 * v0)) / rtb_Saturation1;
(* '<S2>:1:20' CstVelTime=(PositionSP-2*s_acc)/vs; *)
rtb_Saturation := ((rtb_Saturation - x0) - (2.0 * s_acc)) / rtb_Saturation1;
(* '<S2>:1:21' if CstVelTime < 0 *)

IF rtb_Saturation < 0.0 THEN 
    (* '<S2>:1:22' Error = 1; *)
    Error_0 := 1;
ELSE 
    (* '<S2>:1:23' else *)
    (* '<S2>:1:24' Error = 0; *)
    Error_0 := 0;
END_IF;

(* Time periodes, *)
(* '<S2>:1:28' t1=t0+(as/jm); *)
t1_tmp := rtb_Saturation1 / Jerk_Ref;
t1 := t1_tmp + t0;
(* '<S2>:1:29' t2=t1+(as/jm); *)
t2 := t1_tmp + t1;
(* '<S2>:1:30' t3=t2+CstVelTime; *)
t3 := t2 + rtb_Saturation;
(* '<S2>:1:31' t4=t3+(as/jm); *)
t4 := t1_tmp + t3;
(* '<S2>:1:32' t5=t4+(as/jm); *)
Motion_Cycle_Time := t1_tmp + t4;
(* '<S2>:1:33' t6=t5+HoldPositionTime; *)
t6 := Motion_Cycle_Time + t_Hold_Position;
(* '<S2>:1:34' t7=t6+(as/jm); *)
t7 := t1_tmp + t6;
(* '<S2>:1:35' t8=t7+(as/jm); *)
t8 := t1_tmp + t7;
(* '<S2>:1:36' t9=t8+CstVelTime; *)
t9 := t8 + rtb_Saturation;
(* '<S2>:1:37' t10=t9+(as/jm); *)
t10 := t1_tmp + t9;
(* '<S2>:1:38' t11=t10+(as/jm); *)
(* Position and Velocity Constants *)
(* '<S2>:1:40' sh=(v0+(as^2)/(6*jm))*(as/jm); *)
sh := ((sh / (6.0 * Jerk_Ref)) + v0) * t1_tmp;
(* '<S2>:1:41' vh=(vs-v0)/2; *)
vh := vh / 2.0;
(* '<S2>:1:42' s3=s_acc+vs*(t3-t2); *)
s3 := ((t3 - t2) * rtb_Saturation1) + s_acc;
(* '<S2>:1:43' s4=s3+vs*(t4-t3)-jm*((t4-t3)^3)/6; *)
rtb_Saturation := t4 - t3;
s4 := ((rtb_Saturation * rtb_Saturation1) + s3) - ((EXPT(rtb_Saturation, 3.0) * Jerk_Ref) / 6.0);
(* '<S2>:1:44' v4=vs-jm*((t4-t3)^2)/2; *)
v4 := rtb_Saturation1 - (((rtb_Saturation * rtb_Saturation) * Jerk_Ref) / 2.0);
(* '<S2>:1:45' s5=s0+jm*((t5-t4)^3)/6-as*((t5-t4)^2)/2+v4*(t5-t4)+s4; *)
t1_tmp := Motion_Cycle_Time - t4;
rtb_Saturation := (((((EXPT(t1_tmp, 3.0) * Jerk_Ref) / 6.0) + x0) - (((t1_tmp * t1_tmp) * rtb_Saturation1) / 2.0)) + (t1_tmp * v4)) + s4;
(* s6=s5+(s0+v0*(t7-t6)+jm*((t7-t6)^3)/6); *)
(* '<S2>:1:47' s7= s5-(s_acc+vs*(t9-t8)); *)
s7 := rtb_Saturation - (((t9 - t8) * rtb_Saturation1) + s_acc);
(* '<S2>:1:48' s8= s7-(vs*(t10-t9)-jm*((t10-t9)^3)/6); *)
(* s9= s8-(jm*((t11-t10)^3)/6-as*((t11-t10)^2)/2+v4*(t11-t10)); *)
(* Phase0 *)
(* '<S2>:1:51' if  Error == 1 *)

IF Error_0 = 1 THEN 
    (* '<S2>:1:52' s = s0; *)
    rtb_Saturation := x0;
    (* '<S2>:1:53' v = v0; *)
    Position_Ref := v0;
    (* '<S2>:1:54' a = a0; *)
    Acceleration_Ref := 0.0;
    (* '<S2>:1:55' j=j0; *)
    Jerk_Ref := 0.0;
ELSIF (CyclicTime >= 0.0) AND (CyclicTime <= t0) THEN 
    (* '<S2>:1:56' elseif  (t >= 0) &amp;&amp; (t <= t0) *)
    (* '<S2>:1:57' s = s0; *)
    rtb_Saturation := x0;
    (* '<S2>:1:58' v = v0; *)
    Position_Ref := v0;
    (* '<S2>:1:59' a = a0; *)
    Acceleration_Ref := 0.0;
    (* '<S2>:1:60' j=j0; *)
    Jerk_Ref := 0.0;
    (* Phase1 - concave Acc *)
ELSIF (CyclicTime >= t0) AND (CyclicTime <= t1) THEN 
    (* '<S2>:1:62' elseif  (t >= t0) &amp;&amp; (t <= (t1)) *)
    (* '<S2>:1:63' s = s0+v0*(t-t0)+jm*((t-t0)^3)/6; *)
    t1_tmp := CyclicTime - t0;
    rtb_Saturation := ((t1_tmp * v0) + x0) + ((EXPT(t1_tmp, 3.0) * Jerk_Ref) / 6.0);
    (* '<S2>:1:64' v = v0+jm*((t-t0)^2)/2; *)
    Position_Ref := (((t1_tmp * t1_tmp) * Jerk_Ref) / 2.0) + v0;
    (* '<S2>:1:65' a = jm*(t-t0); *)
    Acceleration_Ref := t1_tmp * Jerk_Ref;
    (* '<S2>:1:66' j=jm; *)
    (* Phase2 - convex Acc *)
ELSIF (CyclicTime >= t1) AND (CyclicTime <= t2) THEN 
    (* '<S2>:1:68' elseif (t >= (t1)) &amp;&amp; (t <= (t2)) *)
    (* '<S2>:1:69' s = s0+sh+vh*(t-t1)+as*((t-t1)^2)/2-jm*((t-t1)^3)/6; *)
    t1_tmp := CyclicTime - t1;
    rtb_Saturation := (((t1_tmp * vh) + (x0 + sh)) + (((t1_tmp * t1_tmp) * rtb_Saturation1) / 2.0)) - ((EXPT(t1_tmp, 3.0) * Jerk_Ref) / 6.0);
    (* '<S2>:1:70' v = vh+as*(t-t1)-jm*((t-t1)^2)/2; *)
    Position_Ref := (((CyclicTime - t1) * rtb_Saturation1) + vh) - (((t1_tmp * t1_tmp) * Jerk_Ref) / 2.0);
    (* '<S2>:1:71' a = as-jm*(t-t1); *)
    Acceleration_Ref := rtb_Saturation1 - ((CyclicTime - t1) * Jerk_Ref);
    (* '<S2>:1:72' j = -jm; *)
    Jerk_Ref :=  -Jerk_Ref;
    (* Phase3 - constant velocity *)
ELSIF (CyclicTime >= t2) AND (CyclicTime <= t3) THEN 
    (* '<S2>:1:74' elseif (t >= t2) &amp;&amp; (t <= t3) *)
    (* '<S2>:1:75' s = s0+s_acc+vs*(t-t2); *)
    rtb_Saturation := ((CyclicTime - t2) * rtb_Saturation1) + (x0 + s_acc);
    (* '<S2>:1:76' v = vs; *)
    Position_Ref := rtb_Saturation1;
    (* '<S2>:1:77' a = 0; *)
    Acceleration_Ref := 0.0;
    (* '<S2>:1:78' j = 0; *)
    Jerk_Ref := 0.0;
    (* Phase4 - convex Dec *)
ELSIF (CyclicTime >= t3) AND (CyclicTime <= t4) THEN 
    (* '<S2>:1:80' elseif (t >= t3) &amp;&amp; (t <= t4) *)
    (* '<S2>:1:81' s = s0+s3+vs*(t-t3)-jm*((t-t3)^3)/6; *)
    t1_tmp := CyclicTime - t3;
    rtb_Saturation := ((t1_tmp * rtb_Saturation1) + (x0 + s3)) - ((EXPT(t1_tmp, 3.0) * Jerk_Ref) / 6.0);
    (* '<S2>:1:82' v = vs-jm*((t-t3)^2)/2; *)
    Position_Ref := rtb_Saturation1 - (((t1_tmp * t1_tmp) * Jerk_Ref) / 2.0);
    (* '<S2>:1:83' a = -jm*(t-t3); *)
    Acceleration_Ref := t1_tmp * ( -Jerk_Ref);
    (* '<S2>:1:84' j = -jm; *)
    Jerk_Ref :=  -Jerk_Ref;
    (* Phase5 - concav Dec *)
ELSIF (CyclicTime >= t4) AND (CyclicTime <= Motion_Cycle_Time) THEN 
    (* '<S2>:1:86' elseif (t >= t4) &amp;&amp; (t <= t5) *)
    (* '<S2>:1:87' s = s0+jm*((t-t4)^3)/6-as*((t-t4)^2)/2+v4*(t-t4)+s4; *)
    rtb_Saturation := CyclicTime - t4;
    t1_tmp := CyclicTime - t4;
    rtb_Saturation := (((((EXPT(t1_tmp, 3.0) * Jerk_Ref) / 6.0) + x0) - (((rtb_Saturation * rtb_Saturation) * rtb_Saturation1) / 2.0)) + (t1_tmp * v4)) + s4;
    (* '<S2>:1:88' v = jm*((t-t4)^2)/2-as*(t-t4)+v4; *)
    Position_Ref := ((((t1_tmp * t1_tmp) * Jerk_Ref) / 2.0) - (t1_tmp * rtb_Saturation1)) + v4;
    (* '<S2>:1:89' a = jm*(t-t4)-as; *)
    Acceleration_Ref := (t1_tmp * Jerk_Ref) - rtb_Saturation1;
    (* '<S2>:1:90' j=jm; *)
    (* Phase6 - holding position *)
ELSIF (CyclicTime >= Motion_Cycle_Time) AND (CyclicTime <= t6) THEN 
    (* '<S2>:1:92' elseif (t >= t5) &amp;&amp; (t <= t6) *)
    (* '<S2>:1:93' s = s5; *)
    (* '<S2>:1:94' v = 0; *)
    Position_Ref := 0.0;
    (* '<S2>:1:95' a = 0; *)
    Acceleration_Ref := 0.0;
    (* '<S2>:1:96' j = 0; *)
    Jerk_Ref := 0.0;
    (* Phase7 - concave Dec *)
ELSIF (CyclicTime >= t6) AND (CyclicTime <= t7) THEN 
    (* '<S2>:1:98' elseif (t >= t6) &amp;&amp; (t <= t7) *)
    (* '<S2>:1:99' s = s5-(v0*(t-t6)+jm*((t-t6)^3)/6); *)
    t1_tmp := CyclicTime - t6;
    rtb_Saturation := rtb_Saturation - (((EXPT(t1_tmp, 3.0) * Jerk_Ref) / 6.0) + (t1_tmp * v0));
    (* '<S2>:1:100' v = -(v0+jm*((t-t6)^2)/2); *)
    Position_Ref :=  -((((t1_tmp * t1_tmp) * Jerk_Ref) / 2.0) + v0);
    (* '<S2>:1:101' a = -jm*(t-t6); *)
    Acceleration_Ref := t1_tmp * ( -Jerk_Ref);
    (* '<S2>:1:102' j=-jm; *)
    Jerk_Ref :=  -Jerk_Ref;
    (* Phase8 - convex Dec *)
ELSIF (CyclicTime >= t7) AND (CyclicTime <= t8) THEN 
    (* '<S2>:1:104' elseif (t >= t7) &amp;&amp; (t <= t8) *)
    (* '<S2>:1:105' s = s5-(sh+vh*(t-t7)+as*((t-t7)^2)/2-jm*((t-t7)^3)/6); *)
    t1_tmp := CyclicTime - t7;
    rtb_Saturation := rtb_Saturation - ((((t1_tmp * vh) + sh) + (((t1_tmp * t1_tmp) * rtb_Saturation1) / 2.0)) - ((EXPT(t1_tmp, 3.0) * Jerk_Ref) / 6.0));
    (* '<S2>:1:106' v = -(vh+as*(t-t7)-jm*((t-t7)^2)/2); *)
    Position_Ref :=  -(((t1_tmp * rtb_Saturation1) + vh) - (((t1_tmp * t1_tmp) * Jerk_Ref) / 2.0));
    (* '<S2>:1:107' a = -(as-jm*(t-t7)); *)
    Acceleration_Ref :=  -(rtb_Saturation1 - (t1_tmp * Jerk_Ref));
    (* '<S2>:1:108' j = jm; *)
    (* Phase9 - constant velocity *)
ELSIF (CyclicTime >= t8) AND (CyclicTime <= t9) THEN 
    (* '<S2>:1:110' elseif (t >= t8) &amp;&amp; (t <= t9) *)
    (* '<S2>:1:111' s = s5-(s_acc+vs*(t-t8)); *)
    rtb_Saturation := rtb_Saturation - (((CyclicTime - t8) * rtb_Saturation1) + s_acc);
    (* '<S2>:1:112' v = -vs; *)
    Position_Ref :=  -rtb_Saturation1;
    (* '<S2>:1:113' a = 0; *)
    Acceleration_Ref := 0.0;
    (* '<S2>:1:114' j = 0; *)
    Jerk_Ref := 0.0;
    (* Phase10 - concav Acc *)
ELSIF (CyclicTime >= t9) AND (CyclicTime <= t10) THEN 
    (* '<S2>:1:116' elseif (t >= t9) &amp;&amp; (t <= t10) *)
    (* '<S2>:1:117' s = s7-(vs*(t-t9)-jm*((t-t9)^3)/6); *)
    t1_tmp := CyclicTime - t9;
    rtb_Saturation := s7 - ((t1_tmp * rtb_Saturation1) - ((EXPT(t1_tmp, 3.0) * Jerk_Ref) / 6.0));
    (* '<S2>:1:118' v = -(vs-jm*((t-t9)^2)/2); *)
    Position_Ref :=  -(rtb_Saturation1 - (((t1_tmp * t1_tmp) * Jerk_Ref) / 2.0));
    (* '<S2>:1:119' a = jm*(t-t9); *)
    Acceleration_Ref := t1_tmp * Jerk_Ref;
    (* '<S2>:1:120' j = jm; *)
    (* Phase11 - convex Acc *)
ELSE 
    temp1 := FALSE;

    IF CyclicTime >= t10 THEN 

        IF CyclicTime <= ((rtb_Saturation1 / Jerk_Ref) + t10) THEN 
            (* '<S2>:1:122' elseif (t >= t10) &amp;&amp; (t <= t11) *)
            (* '<S2>:1:123' s = s8-(jm*((t-t10)^3)/6-as*((t-t10)^2)/2+v4*(t-t10)); *)
            t1_tmp := CyclicTime - t10;
            rtb_Saturation := t10 - t9;
            rtb_Saturation := (s7 - ((rtb_Saturation * rtb_Saturation1) - ((EXPT(rtb_Saturation, 3.0) * Jerk_Ref) / 6.0))) - ((((EXPT(t1_tmp, 3.0) * Jerk_Ref) / 6.0) - (((t1_tmp * t1_tmp) * rtb_Saturation1) / 2.0)) + (t1_tmp * v4));
            (* '<S2>:1:124' v = -(jm*((t-t10)^2)/2-as*(t-t10)+v4); *)
            Position_Ref :=  -(((((t1_tmp * t1_tmp) * Jerk_Ref) / 2.0) - (t1_tmp * rtb_Saturation1)) + v4);
            (* '<S2>:1:125' a = -(jm*(t-t10)-as); *)
            Acceleration_Ref :=  -((t1_tmp * Jerk_Ref) - rtb_Saturation1);
            (* '<S2>:1:126' j=-jm; *)
            Jerk_Ref :=  -Jerk_Ref;
            (* Phase12 - hold position *)
        ELSE 
            temp1 := TRUE;
        END_IF;

    ELSE 
        temp1 := TRUE;
    END_IF;


    IF temp1 THEN 
        (* '<S2>:1:128' else *)
        (* '<S2>:1:129' s = s0; *)
        rtb_Saturation := x0;
        (* '<S2>:1:130' v = v0; *)
        Position_Ref := v0;
        (* '<S2>:1:131' a = a0; *)
        Acceleration_Ref := 0.0;
        (* '<S2>:1:132' j = j0; *)
        Jerk_Ref := 0.0;
    END_IF;

END_IF;

(* '<S2>:1:135' if t == 0 *)

IF CyclicTime = 0.0 THEN 
    (* '<S2>:1:136' PositionRef=s0; *)
    rtb_Saturation := x0;
    (* [mm] *)
END_IF;

(* Switch: '<S1>/Switch' *)
(* '<S2>:1:141' InPositionTime=t5; *)
(* [s] *)
(* '<S2>:1:142' VelocityRef=v; *)
(* [mm/s] *)
(* '<S2>:1:143' AccelerationRef=a; *)
(* [mm/s^2] *)
(* '<S2>:1:144' JerkRef=j; *)
(* %[mm/s^3] *)

IF  NOT Enable THEN 
    Position_Ref := v0;
END_IF;

(* End of Switch: '<S1>/Switch' *)


(* Saturate: '<S1>/Saturation2' *)

IF Position_Ref >= 150.0 THEN 
    (* Outport: '<Root>/Velocity_Ref' *)
    Velocity_Ref := 150.0;
ELSIF Position_Ref > -150.0 THEN 
    (* Outport: '<Root>/Velocity_Ref' *)
    Velocity_Ref := Position_Ref;
ELSE 
    (* Outport: '<Root>/Velocity_Ref' *)
    Velocity_Ref := -150.0;
END_IF;

(* End of Saturate: '<S1>/Saturation2' *)


(* Switch: '<S1>/Switch1' incorporates:
 *  Switch: '<S1>/Switch2'
 *  Switch: '<S1>/Switch3' *)

IF Enable THEN 
    Position_Ref := rtb_Saturation;
ELSE 
    Position_Ref := x0;
    (* Outport: '<Root>/Acceleration_Ref' incorporates:
     *  Constant: '<S1>/Constant' *)
    Acceleration_Ref := 0.0;
    (* Outport: '<Root>/Jerk_Ref' incorporates:
     *  Constant: '<S1>/Constant' *)
    Jerk_Ref := 0.0;
END_IF;

(* End of Switch: '<S1>/Switch1' *)


(* Saturate: '<S1>/Saturation3' *)

IF Position_Ref >= 500.0 THEN 
    (* Outport: '<Root>/Position_Ref' *)
    Position_Ref := 500.0;
ELSIF Position_Ref <= 0.0 THEN 
    (* Outport: '<Root>/Position_Ref' *)
    Position_Ref := 0.0;
END_IF;

(* End of Saturate: '<S1>/Saturation3' *)


(* Outport: '<Root>/Error' incorporates:
 *  MATLAB Function: '<S1>/SP_Generator' *)
Error := DINT_TO_LREAL(Error_0);
(* End of Outputs for SubSystem: '<Root>/S_shape_Profile' *)

END_FUNCTION_BLOCK

// IndraMotionMlc1/Application/Subsystem
FUNCTION_BLOCK Subsystem
VAR_INPUT
	In1: LREAL;
END_VAR
VAR_OUTPUT
	Out1: LREAL;
END_VAR
VAR
	frac: LREAL;
	iRght: UDINT;
	iLeft: UDINT;
	bpIdx: UDINT;
	uDLookupTable_tableData: ARRAY[0..10] OF LREAL := [-0.99990920426259511, -0.999329299739067, -0.99505475368673046, -0.9640275800758169, -0.76159415595576485, 0.0, 0.76159415595576485, 0.9640275800758169, 0.99505475368673046, 0.999329299739067, 0.99990920426259511];
	uDLookupTable_bp01Data: ARRAY[0..10] OF LREAL := [-5.0, -4.0, -3.0, -2.0, -1.0, 0.0, 1.0, 2.0, 3.0, 4.0, 5.0];
END_VAR


(* Lookup_n-D: '<S1>/1-D Lookup Table' *)
(* Lookup 1-D
   Search method: 'binary'
   Use previous index: 'off'
   Interpolation method: 'Linear'
   Extrapolation method: 'Linear'
   Use last breakpoint for index at or above upper limit: 'off'
   Remove protection against out-of-range input in generated code: 'off' *)
(* Prelookup - Index and Fraction
   Index Search method: 'binary'
   Extrapolation method: 'Linear'
   Use previous index: 'off'
   Use last breakpoint for index at or above upper limit: 'off'
   Remove protection against out-of-range input in generated code: 'off' *)

IF In1 <= -5.0 THEN 
    iLeft := 0;
    frac := In1 - -5.0;
ELSIF In1 < 5.0 THEN 
    (* Binary Search *)
    bpIdx := 5;
    iLeft := 0;
    iRght := 10;
    WHILE (iRght - iLeft) > 1 DO

        IF In1 < uDLookupTable_bp01Data[bpIdx] THEN 
            iRght := bpIdx;
        ELSE 
            iLeft := bpIdx;
        END_IF;

        bpIdx := DWORD_TO_UDINT(SHR(UDINT_TO_DWORD(iRght + iLeft), 1));
    END_WHILE;
    frac := (In1 - uDLookupTable_bp01Data[iLeft]) / (uDLookupTable_bp01Data[iLeft + 1] - uDLookupTable_bp01Data[iLeft]);
ELSE 
    iLeft := 9;
    frac := In1 - 4.0;
END_IF;

(* Outport: '<Root>/Out1' incorporates:
 *  Lookup_n-D: '<S1>/1-D Lookup Table' *)
(* Interpolation 1-D
   Interpolation method: 'Linear'
   Use last breakpoint for index at or above upper limit: 'off'
   Overflow mode: 'wrapping' *)
Out1 := ((uDLookupTable_tableData[iLeft + 1] - uDLookupTable_tableData[iLeft]) * frac) + uDLookupTable_tableData[iLeft];

END_FUNCTION_BLOCK

// IndraMotionMlc1/Application/Ramp_Profile
FUNCTION_BLOCK Ramp_Profile
VAR_INPUT
	Enable: BOOL;
	x0: LREAL;
	v0: LREAL;
	Position_SP: LREAL;
	Velocity_SP: LREAL;
	t0: LREAL;
	tRamp: LREAL;
	t_Hold_Position: LREAL;
	CyclicTime: LREAL;
END_VAR
VAR_OUTPUT
	Position_Ref: LREAL;
	Velocity_Ref: LREAL;
	Motion_Cycle_Time: LREAL;
	Error: LREAL;
END_VAR
VAR
	Error_0: DINT;
	slopeExt: LREAL;
	tHold: LREAL;
	x1: LREAL;
	x4: LREAL;
	x1_tmp_tmp: LREAL;
	x4_tmp: LREAL;
	x4_tmp_tmp: LREAL;
	x4_tmp_tmp_0: LREAL;
	x4_tmp_tmp_1: LREAL;
	x4_tmp_0: LREAL;
END_VAR


(* Saturate: '<S1>/Saturation3' *)

IF Position_SP >= 500.0 THEN 
    Position_Ref := 500.0;
ELSIF Position_SP > 0.0 THEN 
    Position_Ref := Position_SP;
ELSE 
    Position_Ref := 0.0;
END_IF;

(* End of Saturate: '<S1>/Saturation3' *)


(* Saturate: '<S1>/Saturation2' *)

IF Velocity_SP >= 150.0 THEN 
    Velocity_Ref := 150.0;
ELSIF Velocity_SP > 0.0 THEN 
    Velocity_Ref := Velocity_SP;
ELSE 
    Velocity_Ref := 0.0;
END_IF;

(* End of Saturate: '<S1>/Saturation2' *)


(* MATLAB Function: '<S1>/WaveSignal' *)
(* MATLAB Function 'Ramp_Profile/WaveSignal': '<S2>:1' *)
(* '<S2>:1:2' x_SP = x_ref - x0; *)
(* '<S2>:1:3' vs=v_ref; *)
(* '<S2>:1:4' slopeExt=v0-vs; *)
slopeExt := v0 - Velocity_Ref;
(* '<S2>:1:5' slopeRetr=-vs-v0; *)
(* '<S2>:1:7' as = vs/tRamp; *)
(* '<S2>:1:8' s_acc=(vs^2-v0^2)/as; *)
(* '<S2>:1:10' tHold=(x_SP-s_acc)/vs; *)
tHold := ((Position_Ref - x0) - (((Velocity_Ref * Velocity_Ref) - (v0 * v0)) / (Velocity_Ref / tRamp))) / Velocity_Ref;
(* '<S2>:1:12' if tHold < 0 *)

IF tHold < 0.0 THEN 
    (* '<S2>:1:13' Error = 1; *)
    Error_0 := 1;
ELSE 
    (* '<S2>:1:14' else *)
    (* '<S2>:1:15' Error = 0; *)
    Error_0 := 0;
END_IF;

(* '<S2>:1:18' t1=tRamp; *)
(* '<S2>:1:19' t2=tHold; *)
(* '<S2>:1:20' t3=tRamp; *)
(* '<S2>:1:21' t4=tWait; *)
(* '<S2>:1:22' t5=t1; *)
(* '<S2>:1:23' t6=t2; *)
(* '<S2>:1:24' t7=t3; *)
(* '<S2>:1:26' x = x0; *)
(* '<S2>:1:27' x1 = x0 + v0*((t0+t1)-t0)-(slopeExt/t1)*((t0+t1)-t0)^2/2; *)
x1_tmp_tmp := t0 + tRamp;
x1 := x1_tmp_tmp - t0;
x1 := ((x1 * v0) + x0) - (((slopeExt / tRamp) * (x1 * x1)) / 2.0);
(* '<S2>:1:28' x2 = x1 + vs*((t0+t1+t2)-(t0+t1)); *)
(* '<S2>:1:29' x4 = x_ref - v0*((t0+t1+t2+t3+t4+t5)-(t0+t1+t2+t3+t4))+(slopeRetr/t5)*((t0+t1+t2+t3+t4+t5)-(t0+t1+t2+t3+t4))^2/2; *)
x4_tmp_tmp := x1_tmp_tmp + tHold;
x4_tmp_tmp_0 := x4_tmp_tmp + tRamp;
x4_tmp := x4_tmp_tmp_0 + t_Hold_Position;
x4_tmp_tmp_1 := x4_tmp + tRamp;
x4 := x4_tmp_tmp_1 - x4_tmp;
x4_tmp_0 := (( -Velocity_Ref) - v0) / tRamp;
x4 := (Position_Ref - (x4 * v0)) + ((x4_tmp_0 * (x4 * x4)) / 2.0);
(* '<S2>:1:30' x5 = x4-vs*((t0+t1+t2+t3+t4+t5+t6)-(t0+t1+t2+t3+t4+t5)); *)
(* '<S2>:1:32' if Error == 1 *)

IF Error_0 = 1 THEN 
    (* '<S2>:1:33' x = x0; *)
    Position_Ref := x0;
    (* '<S2>:1:34' v = v0; *)
    Velocity_Ref := v0;
ELSIF (CyclicTime >= 0.0) AND (CyclicTime < t0) THEN 
    (* '<S2>:1:35' elseif t>=0 &amp;&amp; t<t0 *)
    (* '<S2>:1:36' x = x0; *)
    Position_Ref := x0;
    (* '<S2>:1:37' v = v0; *)
    Velocity_Ref := v0;
ELSIF (CyclicTime >= t0) AND (CyclicTime < x1_tmp_tmp) THEN 
    (* '<S2>:1:38' elseif t>=t0 &amp;&amp; t<(t0+t1) *)
    (* '<S2>:1:39' x = x0 + v0*(t-t0)-(slopeExt/t1)*(t-t0)^2/2; *)
    x4_tmp_tmp_1 := CyclicTime - t0;
    Position_Ref := ((x4_tmp_tmp_1 * v0) + x0) - (((slopeExt / tRamp) * (x4_tmp_tmp_1 * x4_tmp_tmp_1)) / 2.0);
    (* '<S2>:1:40' v = v0-(slopeExt/t1)*(t-t0); *)
    Velocity_Ref := v0 - ((slopeExt / tRamp) * x4_tmp_tmp_1);
ELSIF (CyclicTime >= x1_tmp_tmp) AND (CyclicTime < x4_tmp_tmp) THEN 
    (* '<S2>:1:41' elseif t>=(t0+t1) &amp;&amp; t<(t0+t1+t2) *)
    (* '<S2>:1:42' x = x1 + vs*(t-(t0+t1)); *)
    Position_Ref := ((CyclicTime - x1_tmp_tmp) * Velocity_Ref) + x1;
    (* '<S2>:1:43' v = vs; *)
ELSIF (CyclicTime >= x4_tmp_tmp) AND (CyclicTime < x4_tmp_tmp_0) THEN 
    (* '<S2>:1:44' elseif t>=(t0+t1+t2) &amp;&amp; t<(t0+t1+t2+t3) *)
    (* '<S2>:1:45' x = x2+vs*(t-(t0+t1+t2))+(slopeExt/t3)*(t-(t0+t1+t2))^2/2; *)
    x4_tmp_tmp_1 := CyclicTime - x4_tmp_tmp;
    slopeExt := slopeExt / tRamp;
    Position_Ref := ((((x4_tmp_tmp - x1_tmp_tmp) * Velocity_Ref) + x1) + (x4_tmp_tmp_1 * Velocity_Ref)) + ((slopeExt * (x4_tmp_tmp_1 * x4_tmp_tmp_1)) / 2.0);
    (* '<S2>:1:46' v = vs+(slopeExt/t3)*(t-(t0+t1+t2)); *)
    Velocity_Ref := (x4_tmp_tmp_1 * slopeExt) + Velocity_Ref;
ELSIF (CyclicTime >= x4_tmp_tmp_0) AND (CyclicTime < x4_tmp) THEN 
    (* '<S2>:1:47' elseif t>=(t0+t1+t2+t3) &amp;&amp; t<(t0+t1+t2+t3+t4) *)
    (* '<S2>:1:48' x = x_ref; *)
    (* '<S2>:1:49' v = v0; *)
    Velocity_Ref := v0;
ELSIF (CyclicTime >= x4_tmp) AND (CyclicTime < x4_tmp_tmp_1) THEN 
    (* '<S2>:1:50' elseif t>=(t0+t1+t2+t3+t4) &amp;&amp; t<(t0+t1+t2+t3+t4+t5) *)
    (* '<S2>:1:51' x = x_ref - v0*(t-(t0+t1+t2+t3+t4))+(slopeRetr/t5)*(t-(t0+t1+t2+t3+t4))^2/2; *)
    x1_tmp_tmp := CyclicTime - x4_tmp;
    Position_Ref := (Position_Ref - (x1_tmp_tmp * v0)) + ((x4_tmp_0 * (x1_tmp_tmp * x1_tmp_tmp)) / 2.0);
    (* '<S2>:1:52' v = v0+(slopeRetr/t5)*(t-(t0+t1+t2+t3+t4)); *)
    Velocity_Ref := (x1_tmp_tmp * x4_tmp_0) + v0;
ELSE 
    slopeExt := x4_tmp_tmp_1 + tHold;

    IF (CyclicTime >= x4_tmp_tmp_1) AND (CyclicTime < slopeExt) THEN 
        (* '<S2>:1:53' elseif t>=(t0+t1+t2+t3+t4+t5) &amp;&amp; t<(t0+t1+t2+t3+t4+t5+t6) *)
        (* '<S2>:1:54' x = x4-vs*(t-(t0+t1+t2+t3+t4+t5)); *)
        Position_Ref := x4 - ((CyclicTime - x4_tmp_tmp_1) * Velocity_Ref);
        (* '<S2>:1:55' v = -vs; *)
        Velocity_Ref :=  -Velocity_Ref;
    ELSIF (CyclicTime >= slopeExt) AND (CyclicTime < (slopeExt + tRamp)) THEN 
        (* '<S2>:1:56' elseif t>=(t0+t1+t2+t3+t4+t5+t6) &amp;&amp; t<(t0+t1+t2+t3+t4+t5+t6+t7) *)
        (* '<S2>:1:57' x = x5-vs*(t-(t0+t1+t2+t3+t4+t5+t6))-(slopeRetr/t3)*(t-(t0+t1+t2+t3+t4+t5+t6))^2/2; *)
        x1_tmp_tmp := CyclicTime - slopeExt;
        Position_Ref := ((x4 - ((slopeExt - x4_tmp_tmp_1) * Velocity_Ref)) - (x1_tmp_tmp * Velocity_Ref)) - ((x4_tmp_0 * (x1_tmp_tmp * x1_tmp_tmp)) / 2.0);
        (* '<S2>:1:58' v = -vs-(slopeRetr/t3)*(t-(t0+t1+t2+t3+t4+t5+t6)); *)
        Velocity_Ref := ( -Velocity_Ref) - (x1_tmp_tmp * x4_tmp_0);
    ELSE 
        (* '<S2>:1:59' else *)
        (* '<S2>:1:60' x = x0; *)
        Position_Ref := x0;
        (* '<S2>:1:61' v = v0; *)
        Velocity_Ref := v0;
    END_IF;

END_IF;

(* Switch: '<S1>/Switch' incorporates:
 *  Switch: '<S1>/Switch1' *)
(* '<S2>:1:64' T = t0+t1+t2+t3+t4+t5+t6+t7; *)

IF  NOT Enable THEN 
    Velocity_Ref := v0;
    Position_Ref := x0;
END_IF;

(* End of Switch: '<S1>/Switch' *)


(* Saturate: '<S1>/Saturation' *)

IF Velocity_Ref >= 150.0 THEN 
    Velocity_Ref := 150.0;
ELSIF Velocity_Ref <= -150.0 THEN 
    Velocity_Ref := -150.0;
END_IF;

(* End of Saturate: '<S1>/Saturation' *)


(* Saturate: '<S1>/Saturation1' *)

IF Position_Ref >= 500.0 THEN 
    Position_Ref := 500.0;
ELSIF Position_Ref <= 0.0 THEN 
    Position_Ref := 0.0;
END_IF;

(* End of Saturate: '<S1>/Saturation1' *)


(* Outport: '<Root>/Motion_Cycle_Time' incorporates:
 *  MATLAB Function: '<S1>/WaveSignal' *)
Motion_Cycle_Time := ((((((t0 + tRamp) + tHold) + tRamp) + t_Hold_Position) + tRamp) + tHold) + tRamp;
(* Outport: '<Root>/Error' incorporates:
 *  MATLAB Function: '<S1>/WaveSignal' *)
Error := DINT_TO_LREAL(Error_0);

END_FUNCTION_BLOCK

// IndraMotionMlc1/Application/VCC_Pos_Step
FUNCTION_BLOCK VCC_Pos_Step
VAR_INPUT
	Enable: BOOL;
	x0: LREAL;
	xSP: LREAL;
	t0: LREAL;
	tHold: LREAL;
	Clock: LREAL;
END_VAR
VAR_OUTPUT
	xC_ref: LREAL;
END_VAR
VAR
END_VAR


(* MATLAB Function: '<S1>/StepFunction' *)
(* MATLAB Function 'VCC_Pos_Step/StepFunction': '<S2>:1' *)
(* '<S2>:1:4' if t>=0 &amp;&amp; t<t0 *)

IF (Clock >= 0.0) AND (Clock < t0) THEN 
    (* '<S2>:1:5' y = x0; *)
    xC_ref := x0;
ELSIF (Clock >= t0) AND (Clock < (t0 + tHold)) THEN 
    (* '<S2>:1:6' elseif t>=(t0) &amp;&amp; t<(t0+t1) *)
    (* '<S2>:1:7' y = x_SP; *)
    xC_ref := xSP;
ELSE 
    (* '<S2>:1:8' else *)
    (* '<S2>:1:9' y = x0; *)
    xC_ref := x0;
END_IF;

(* End of MATLAB Function: '<S1>/StepFunction' *)


(* Switch: '<S1>/Switch' *)

IF  NOT Enable THEN 
    (* Outport: '<Root>/xC_ref' incorporates:
     *  Constant: '<S1>/Constant' *)
    xC_ref := 0.0;
END_IF;

(* End of Switch: '<S1>/Switch' *)

END_FUNCTION_BLOCK

// IndraMotionMlc1/Application/SCC_SinProfile
FUNCTION_BLOCK SCC_SinProfile
VAR_INPUT
	Enable: BOOL;
	x0: LREAL;
	v0: LREAL;
	xC_SP: LREAL;
	T: LREAL;
	Clock: LREAL;
END_VAR
VAR_OUTPUT
	xC: LREAL;
	vC: LREAL;
END_VAR
VAR
	A: LREAL;
	xC_tmp: LREAL;
END_VAR


(* MATLAB Function: '<S1>/WaveSignal' *)
(* MATLAB Function 'SCC_SinProfile/WaveSignal': '<S2>:1' *)
(* '<S2>:1:3' A=xC_SP/2; *)
A := xC_SP / 2.0;
(* Switch: '<S1>/Switch' incorporates:
 *  Switch: '<S1>/Switch1' *)
(* '<S2>:1:5' x0=x0+A; *)
(* '<S2>:1:6' v0=v0; *)
(* '<S2>:1:8' x = x0+A*cos(2*pi*(1/Ts)*t+phi); *)
(* '<S2>:1:9' dx = v0-2*pi*A*(1/Ts)*sin(2*pi*(1/Ts)*t+phi); *)

IF Enable THEN 
    (* MATLAB Function: '<S1>/WaveSignal' incorporates:
     *  Constant: '<S1>/Constant1' *)
    xC_tmp := (((1.0 / T) * 6.2831853071795862) * Clock) + 3.1415926535897931;
    (* Outport: '<Root>/xC' incorporates:
     *  MATLAB Function: '<S1>/WaveSignal' *)
    xC := (COS(xC_tmp) * A) + (x0 + A);
    (* Outport: '<Root>/vC' incorporates:
     *  MATLAB Function: '<S1>/WaveSignal' *)
    vC := v0 - (SIN(xC_tmp) * ((6.2831853071795862 * A) * (1.0 / T)));
ELSE 
    (* Outport: '<Root>/xC' incorporates:
     *  Constant: '<S1>/Constant' *)
    xC := 0.0;
    (* Outport: '<Root>/vC' incorporates:
     *  Constant: '<S1>/Constant' *)
    vC := 0.0;
END_IF;

(* End of Switch: '<S1>/Switch' *)

END_FUNCTION_BLOCK

// IndraMotionMlc1/Application/SCC_Vel_AD
FUNCTION_BLOCK SCC_Vel_AD
VAR_INPUT
	ssMethodType: SINT;
	Enable: BOOL;
	usDelay: LREAL;
	HPF_Num1: LREAL;
	HPF_Num2: LREAL;
	HPF_Den1: LREAL;
	HPF_Den2: LREAL;
	xC_mm: LREAL;
END_VAR
VAR_OUTPUT
	uAD: LREAL;
END_VAR
VAR
	rtb_Compare: BOOL;
	rtb_TSamp: LREAL;
	rtb_Diff: LREAL;
	rtb_Switch5: LREAL;
	HP_Filter_states: LREAL;
	UD_DSTATE: LREAL;
	Integrator_PrevResetState: SINT;
	Integrator_IC_LOADING: USINT;
	Integrator_DSTATE: LREAL;
	VectorConcatenate1: ARRAY[0..1] OF LREAL;
	VectorConcatenate: ARRAY[0..1] OF LREAL;
	Probe: ARRAY[0..1] OF LREAL;
END_VAR



CASE ssMethodType OF
    0: 
        (* Start for Probe: '<S4>/Probe' *)
        Probe[0] := 0.001;
        Probe[1] := 0.0;
        (* InitializeConditions for UnitDelay: '<S2>/UD'
         *
         * Block description for '<S2>/UD':
         *  
         *  Store in Global RAM *)
        UD_DSTATE := 0.0;
        (* InitializeConditions for DiscreteIntegrator: '<S8>/Integrator' *)
        Integrator_IC_LOADING := 1;
        Integrator_PrevResetState := 0;
        (* InitializeConditions for DiscreteTransferFcn: '<S1>/HP_Filter' *)
        HP_Filter_states := 0.0;
    1: 
        (* RelationalOperator: '<S6>/Compare' incorporates:
         *  Constant: '<S4>/Time constant'
         *  Constant: '<S6>/Constant'
         *  Sum: '<S4>/Sum1' *)
        rtb_Compare := (0.1 - Probe[0]) <= 0.0;
        (* SampleTimeMath: '<S2>/TSamp' incorporates:
         *  Gain: '<S1>/Gain'
         *
         * About '<S2>/TSamp':
         *  y = u * K where K = 1 / ( w * Ts ) *)
        rtb_TSamp := (0.001 * xC_mm) * 1000.0;
        (* Sum: '<S2>/Diff' incorporates:
         *  UnitDelay: '<S2>/UD'
         *
         * Block description for '<S2>/Diff':
         *  
         *  Add in CPU
         *
         * Block description for '<S2>/UD':
         *  
         *  Store in Global RAM *)
        rtb_Diff := rtb_TSamp - UD_DSTATE;
        (* DiscreteIntegrator: '<S8>/Integrator' *)

        IF Integrator_IC_LOADING <> 0 THEN 
            Integrator_DSTATE := rtb_Diff;

            IF Integrator_DSTATE >= 0.175 THEN 
                Integrator_DSTATE := 0.175;
            ELSIF Integrator_DSTATE <= -0.175 THEN 
                Integrator_DSTATE := -0.175;
            END_IF;

        END_IF;


        IF rtb_Compare OR (Integrator_PrevResetState <> 0) THEN 
            Integrator_DSTATE := rtb_Diff;

            IF Integrator_DSTATE >= 0.175 THEN 
                Integrator_DSTATE := 0.175;
            ELSIF Integrator_DSTATE <= -0.175 THEN 
                Integrator_DSTATE := -0.175;
            END_IF;

        END_IF;


        IF Integrator_DSTATE >= 0.175 THEN 
            Integrator_DSTATE := 0.175;
        ELSIF Integrator_DSTATE <= -0.175 THEN 
            Integrator_DSTATE := -0.175;
        END_IF;

        (* Switch: '<S1>/Switch5' incorporates:
         *  Constant: '<S1>/Constant3'
         *  DiscreteIntegrator: '<S8>/Integrator' *)

        IF usDelay > 2.0 THEN 
            rtb_Switch5 := Integrator_DSTATE;
        ELSE 
            rtb_Switch5 := 0.0;
        END_IF;

        (* End of Switch: '<S1>/Switch5' *)
        

        (* SignalConversion: '<S1>/ConcatBufferAtVector ConcatenateIn1' *)
        VectorConcatenate[0] := HPF_Num1;
        (* SignalConversion: '<S1>/ConcatBufferAtVector ConcatenateIn2' *)
        VectorConcatenate[1] := HPF_Num2;
        (* SignalConversion: '<S1>/ConcatBufferAtVector Concatenate1In1' *)
        VectorConcatenate1[0] := HPF_Den1;
        (* SignalConversion: '<S1>/ConcatBufferAtVector Concatenate1In2' *)
        VectorConcatenate1[1] := HPF_Den2;
        (* DiscreteTransferFcn: '<S1>/HP_Filter' *)
        rtb_Switch5 := rtb_Switch5 - (VectorConcatenate1[1] * HP_Filter_states);
        uAD := (VectorConcatenate[0] * rtb_Switch5) + (VectorConcatenate[1] * HP_Filter_states);
        (* Switch: '<S1>/Switch2' incorporates:
         *  Constant: '<S1>/Constant' *)

        IF Enable THEN 
            (* Switch: '<S1>/Switch1' incorporates:
             *  Constant: '<S1>/Constant' *)

            IF usDelay <= 2.0 THEN 
                uAD := 0.0;
            END_IF;

            (* End of Switch: '<S1>/Switch1' *)
        ELSE 
            uAD := 0.0;
        END_IF;

        (* End of Switch: '<S1>/Switch2' *)
        

        (* Saturate: '<S1>/Saturation5' *)

        IF uAD >= 3600.0 THEN 
            uAD := 3600.0;
        ELSIF uAD <= -3600.0 THEN 
            uAD := -3600.0;
        END_IF;

        (* End of Saturate: '<S1>/Saturation5' *)
        

        (* Update for UnitDelay: '<S2>/UD'
         *
         * Block description for '<S2>/UD':
         *  
         *  Store in Global RAM *)
        UD_DSTATE := rtb_TSamp;
        (* Update for DiscreteIntegrator: '<S8>/Integrator' incorporates:
         *  Constant: '<S4>/Time constant'
         *  MinMax: '<S4>/Max'
         *  Product: '<S3>/1//T'
         *  Sum: '<S3>/Sum1' *)
        Integrator_IC_LOADING := 0;
        Integrator_DSTATE := (((1.0 / MAX(Probe[0], 0.1)) * (rtb_Diff - Integrator_DSTATE)) * 0.001) + Integrator_DSTATE;

        IF Integrator_DSTATE >= 0.175 THEN 
            Integrator_DSTATE := 0.175;
        ELSIF Integrator_DSTATE <= -0.175 THEN 
            Integrator_DSTATE := -0.175;
        END_IF;


        IF rtb_Compare THEN 
            Integrator_PrevResetState := 1;
        ELSE 
            Integrator_PrevResetState := 0;
        END_IF;

        (* End of Update for DiscreteIntegrator: '<S8>/Integrator' *)
        

        (* Update for DiscreteTransferFcn: '<S1>/HP_Filter' *)
        HP_Filter_states := rtb_Switch5;
END_CASE;

END_FUNCTION_BLOCK

// IndraMotionMlc1/Application/SCC_AD_Iq
FUNCTION_BLOCK SCC_AD_Iq
VAR_INPUT
	ssMethodType: SINT;
	Enable: BOOL;
	usDelay: LREAL;
	kQf: LREAL;
	HPF_Num1: LREAL;
	HPF_Num2: LREAL;
	HPF_Den1: LREAL;
	HPF_Den2: LREAL;
	Reset: BOOL;
	Iq: LREAL;
END_VAR
VAR_OUTPUT
	uPF: LREAL;
END_VAR
VAR
	HP_Filter_tmp: LREAL;
	VectorConcatenate: ARRAY[0..1] OF LREAL;
	VectorConcatenate1: ARRAY[0..1] OF LREAL;
	HP_Filter_states: LREAL;
END_VAR



CASE ssMethodType OF
    0: 
        (* InitializeConditions for DiscreteTransferFcn: '<S1>/HP_Filter' *)
        HP_Filter_states := 0.0;
    1: 
        (* SignalConversion: '<S1>/ConcatBufferAtVector ConcatenateIn1' *)
        VectorConcatenate[0] := HPF_Num1;
        (* SignalConversion: '<S1>/ConcatBufferAtVector ConcatenateIn2' *)
        VectorConcatenate[1] := HPF_Num2;
        (* SignalConversion: '<S1>/ConcatBufferAtVector Concatenate1In1' *)
        VectorConcatenate1[0] := HPF_Den1;
        (* SignalConversion: '<S1>/ConcatBufferAtVector Concatenate1In2' *)
        VectorConcatenate1[1] := HPF_Den2;
        (* DiscreteTransferFcn: '<S1>/HP_Filter' *)

        IF Reset THEN 
            HP_Filter_states := 0.0;
        END_IF;

        HP_Filter_tmp := Iq - (VectorConcatenate1[1] * HP_Filter_states);
        (* Switch: '<S1>/Switch2' incorporates:
         *  Constant: '<S1>/Constant' *)

        IF Enable THEN 
            (* Switch: '<S1>/Switch1' incorporates:
             *  Constant: '<S1>/Constant'
             *  DiscreteTransferFcn: '<S1>/HP_Filter'
             *  Product: '<S1>/Product' *)

            IF usDelay > 2.0 THEN 
                uPF := ((VectorConcatenate[0] * HP_Filter_tmp) + (VectorConcatenate[1] * HP_Filter_states)) * kQf;
            ELSE 
                uPF := 0.0;
            END_IF;

            (* End of Switch: '<S1>/Switch1' *)
        ELSE 
            uPF := 0.0;
        END_IF;

        (* End of Switch: '<S1>/Switch2' *)
        

        (* Saturate: '<S1>/Saturation5' *)

        IF uPF >= 3600.0 THEN 
            uPF := 3600.0;
        ELSIF uPF <= -3600.0 THEN 
            uPF := -3600.0;
        END_IF;

        (* End of Saturate: '<S1>/Saturation5' *)
        

        (* Update for DiscreteTransferFcn: '<S1>/HP_Filter' *)
        HP_Filter_states := HP_Filter_tmp;
END_CASE;

END_FUNCTION_BLOCK

// IndraMotionMlc1/Application/SCC_HPPF1
FUNCTION_BLOCK SCC_HPPF1
VAR_INPUT
	ssMethodType: SINT;
	Enable: BOOL;
	usDelay: LREAL;
	kQf: LREAL;
	HPF_Num1: LREAL;
	HPF_Num2: LREAL;
	HPF_Den1: LREAL;
	HPF_Den2: LREAL;
	Reset: BOOL;
	pA_bar: LREAL;
	pB_bar: LREAL;
END_VAR
VAR_OUTPUT
	uPF: LREAL;
END_VAR
VAR
	tempOutEvent: DINT;
	rtb_Switch3: LREAL;
	i0_ZCFCN_d_FALLING: ZCFCN_d_FALLING;
	VectorConcatenate: ARRAY[0..1] OF LREAL;
	VectorConcatenate1: ARRAY[0..1] OF LREAL;
	pp: LREAL;
	pr: LREAL;
	HP_Filter_states: LREAL;
	Subsystem2_Trig_ZCE: USINT := 3;
END_VAR



CASE ssMethodType OF
    0: 
        (* InitializeConditions for DiscreteTransferFcn: '<S1>/HP_Filter' *)
        HP_Filter_states := 0.0;
        (* SystemInitialize for Triggered SubSystem: '<S1>/Subsystem2' *)
        (* SystemInitialize for Outport: '<S2>/pp0' *)
        pp := 0.0;
        (* SystemInitialize for Outport: '<S2>/pr0' *)
        pr := 0.0;
        (* End of SystemInitialize for SubSystem: '<S1>/Subsystem2' *)
    1: 
        (* Switch: '<S1>/Switch3' incorporates:
         *  Constant: '<S1>/Constant1'
         *  Constant: '<S1>/Constant2' *)

        IF usDelay > 0.0 THEN 
            rtb_Switch3 := 0.0;
        ELSE 
            rtb_Switch3 := 1.0;
        END_IF;

        (* End of Switch: '<S1>/Switch3' *)
        

        (* Outputs for Triggered SubSystem: '<S1>/Subsystem2' incorporates:
         *  TriggerPort: '<S2>/Trigger' *)
        i0_ZCFCN_d_FALLING(u0 := Subsystem2_Trig_ZCE, u1 := rtb_Switch3);
        tempOutEvent := i0_ZCFCN_d_FALLING.y0;
        Subsystem2_Trig_ZCE := i0_ZCFCN_d_FALLING.y1;

        IF tempOutEvent <> 0 THEN 
            (* Inport: '<S2>/pp' *)
            pp := pA_bar;
            (* Inport: '<S2>/pr' *)
            pr := pB_bar;
        END_IF;

        (* End of Outputs for SubSystem: '<S1>/Subsystem2' *)
        

        (* SignalConversion: '<S1>/ConcatBufferAtVector ConcatenateIn1' *)
        VectorConcatenate[0] := HPF_Num1;
        (* SignalConversion: '<S1>/ConcatBufferAtVector ConcatenateIn2' *)
        VectorConcatenate[1] := HPF_Num2;
        (* SignalConversion: '<S1>/ConcatBufferAtVector Concatenate1In1' *)
        VectorConcatenate1[0] := HPF_Den1;
        (* SignalConversion: '<S1>/ConcatBufferAtVector Concatenate1In2' *)
        VectorConcatenate1[1] := HPF_Den2;
        (* DiscreteTransferFcn: '<S1>/HP_Filter' incorporates:
         *  Gain: '<S1>/Gain'
         *  Gain: '<S1>/Gain3'
         *  Gain: '<S1>/muC'
         *  Sum: '<S1>/Add'
         *  Sum: '<S1>/Subtract2'
         *  Sum: '<S1>/Subtract3' *)

        IF Reset THEN 
            HP_Filter_states := 0.0;
        END_IF;

        rtb_Switch3 := (((pA_bar - pp) * 100000.0) - (((pB_bar - pr) * 100000.0) * 0.7101)) - (VectorConcatenate1[1] * HP_Filter_states);
        (* Switch: '<S1>/Switch2' incorporates:
         *  Constant: '<S1>/Constant' *)

        IF Enable THEN 
            (* Switch: '<S1>/Switch1' incorporates:
             *  Constant: '<S1>/Constant'
             *  DiscreteTransferFcn: '<S1>/HP_Filter'
             *  Product: '<S1>/Product' *)

            IF usDelay > 2.0 THEN 
                uPF := ((VectorConcatenate[0] * rtb_Switch3) + (VectorConcatenate[1] * HP_Filter_states)) * kQf;
            ELSE 
                uPF := 0.0;
            END_IF;

            (* End of Switch: '<S1>/Switch1' *)
        ELSE 
            uPF := 0.0;
        END_IF;

        (* End of Switch: '<S1>/Switch2' *)
        

        (* Saturate: '<S1>/Saturation5' *)

        IF uPF >= 3600.0 THEN 
            uPF := 3600.0;
        ELSIF uPF <= -3600.0 THEN 
            uPF := -3600.0;
        END_IF;

        (* End of Saturate: '<S1>/Saturation5' *)
        

        (* Update for DiscreteTransferFcn: '<S1>/HP_Filter' *)
        HP_Filter_states := rtb_Switch3;
END_CASE;

END_FUNCTION_BLOCK

// IndraMotionMlc1/Application/ZCFCN_d_FALLING
FUNCTION_BLOCK ZCFCN_d_FALLING
VAR_INPUT
	u0: USINT;
	u1: LREAL;
END_VAR
VAR_OUTPUT
	y0: DINT;
	y1: USINT;
END_VAR
VAR
	falling: BOOL;
	temp1: BOOL;
	temp2: BOOL;
END_VAR


temp1 := FALSE;

IF u1 > 0.0 THEN 
    y1 := 1;
ELSIF u1 < 0.0 THEN 
    y1 := 2;
ELSE 
    y1 := 0;
END_IF;

temp2 := FALSE;

IF u0 = 1 THEN 

    IF y1 = 0 THEN 
        falling := TRUE;
    ELSIF y1 = 2 THEN 
        falling := TRUE;
    ELSE 
        temp2 := TRUE;
    END_IF;

ELSE 
    temp2 := TRUE;
END_IF;


IF temp2 THEN 

    IF u0 = 0 THEN 

        IF y1 = 2 THEN 
            falling := TRUE;
        ELSE 
            temp1 := TRUE;
        END_IF;

    ELSE 
        temp1 := TRUE;
    END_IF;

END_IF;


IF temp1 THEN 

    IF u0 = 100 THEN 

        IF y1 = 2 THEN 
            falling := TRUE;
        ELSE 
            falling := FALSE;
        END_IF;

    ELSE 
        falling := FALSE;
    END_IF;

END_IF;


IF falling THEN 
    y0 := -1;
ELSE 
    y0 := 0;
END_IF;


IF (u0 = 1) AND (y1 = 0) THEN 
    y1 := 101;
END_IF;

END_FUNCTION_BLOCK

// IndraMotionMlc1/Application/SCC_LPPF
FUNCTION_BLOCK SCC_LPPF
VAR_INPUT
	ssMethodType: SINT;
	Enable1: BOOL;
	kQf1: LREAL;
	HPF_Num1: LREAL;
	HPF_Den1: LREAL;
	HPF_Den2: LREAL;
	pAsimbar1: LREAL;
	pBsimbar1: LREAL;
	Clock: LREAL;
	uEM: LREAL;
END_VAR
VAR_OUTPUT
	uPF1: LREAL;
END_VAR
VAR
	tempOutEvent: DINT;
	rtb_Switch3: LREAL;
	i0_ZCFCN_d_FALLING: ZCFCN_d_FALLING;
	VectorConcatenate1: ARRAY[0..1] OF LREAL;
	pp: LREAL;
	pr: LREAL;
	HP_Filter_states: LREAL;
	Subsystem_Trig_ZCE: USINT := 3;
END_VAR



CASE ssMethodType OF
    0: 
        (* InitializeConditions for DiscreteTransferFcn: '<S1>/HP_Filter' *)
        HP_Filter_states := 0.0;
        (* SystemInitialize for Triggered SubSystem: '<S1>/Subsystem' *)
        (* SystemInitialize for Outport: '<S2>/pp0' *)
        pp := 0.0;
        (* SystemInitialize for Outport: '<S2>/pr0' *)
        pr := 0.0;
        (* End of SystemInitialize for SubSystem: '<S1>/Subsystem' *)
    1: 
        (* SignalConversion: '<S1>/ConcatBufferAtVector Concatenate1In1' *)
        VectorConcatenate1[0] := HPF_Den1;
        (* SignalConversion: '<S1>/ConcatBufferAtVector Concatenate1In2' *)
        VectorConcatenate1[1] := HPF_Den2;
        (* Switch: '<S1>/Switch3' incorporates:
         *  Abs: '<S1>/Abs'
         *  Constant: '<S1>/Constant1'
         *  Constant: '<S1>/Constant2' *)

        IF ABS(uEM) > 1.0 THEN 
            rtb_Switch3 := 0.0;
        ELSE 
            rtb_Switch3 := 1.0;
        END_IF;

        (* End of Switch: '<S1>/Switch3' *)
        

        (* Outputs for Triggered SubSystem: '<S1>/Subsystem' incorporates:
         *  TriggerPort: '<S2>/Trigger' *)
        i0_ZCFCN_d_FALLING(u0 := Subsystem_Trig_ZCE, u1 := rtb_Switch3);
        tempOutEvent := i0_ZCFCN_d_FALLING.y0;
        Subsystem_Trig_ZCE := i0_ZCFCN_d_FALLING.y1;

        IF tempOutEvent <> 0 THEN 
            (* Inport: '<S2>/pp' *)
            pp := pAsimbar1;
            (* Inport: '<S2>/pr' *)
            pr := pBsimbar1;
        END_IF;

        (* End of Outputs for SubSystem: '<S1>/Subsystem' *)
        

        (* Switch: '<S1>/Switch4' incorporates:
         *  Constant: '<S1>/Constant3' *)

        IF Enable1 THEN 
            (* Switch: '<S1>/Switch5' incorporates:
             *  Constant: '<S1>/Constant3'
             *  DiscreteTransferFcn: '<S1>/HP_Filter'
             *  Product: '<S1>/Product1' *)

            IF Clock > 0.01 THEN 
                uPF1 := (HPF_Num1 * HP_Filter_states) * kQf1;
            ELSE 
                uPF1 := 0.0;
            END_IF;

            (* End of Switch: '<S1>/Switch5' *)
        ELSE 
            uPF1 := 0.0;
        END_IF;

        (* End of Switch: '<S1>/Switch4' *)
        

        (* Saturate: '<S1>/Saturation1' *)

        IF uPF1 >= 3600.0 THEN 
            uPF1 := 3600.0;
        ELSIF uPF1 <= -3600.0 THEN 
            uPF1 := -3600.0;
        END_IF;

        (* End of Saturate: '<S1>/Saturation1' *)
        

        (* Update for DiscreteTransferFcn: '<S1>/HP_Filter' incorporates:
         *  Gain: '<S1>/Gain1'
         *  Gain: '<S1>/Gain2'
         *  Gain: '<S1>/muC1'
         *  Sum: '<S1>/Add1'
         *  Sum: '<S1>/Subtract'
         *  Sum: '<S1>/Subtract1' *)
        HP_Filter_states := (((pAsimbar1 - pp) * 100000.0) - (((pBsimbar1 - pr) * 100000.0) * 0.7101)) - (VectorConcatenate1[1] * HP_Filter_states);
END_CASE;

END_FUNCTION_BLOCK

// IndraMotionMlc1/Application/SCC_DPF
FUNCTION_BLOCK SCC_DPF
VAR_INPUT
	ssMethodType: SINT;
	Enable: BOOL;
	kQf: LREAL;
	HPF_Num1: LREAL;
	pAsimbar: LREAL;
	pBsimbar: LREAL;
	Clock: LREAL;
	uEM: LREAL;
END_VAR
VAR_OUTPUT
	uPF: LREAL;
END_VAR
VAR
	tempOutEvent: DINT;
	rtb_Switch1: DINT;
	i0_ZCFCN_d_FALLING: ZCFCN_d_FALLING;
	pp: LREAL;
	pr: LREAL;
	Subsystem_Trig_ZCE: USINT := 3;
END_VAR



CASE ssMethodType OF
    0: 
        (* SystemInitialize for Triggered SubSystem: '<S1>/Subsystem' *)
        (* SystemInitialize for Outport: '<S2>/pp0' *)
        pp := 0.0;
        (* SystemInitialize for Outport: '<S2>/pr0' *)
        pr := 0.0;
        (* End of SystemInitialize for SubSystem: '<S1>/Subsystem' *)
    1: 
        (* Switch: '<S1>/Switch1' incorporates:
         *  Abs: '<S1>/Abs'
         *  Constant: '<S1>/Constant1'
         *  Constant: '<S1>/Constant2' *)

        IF ABS(uEM) > 1.0 THEN 
            rtb_Switch1 := 0;
        ELSE 
            rtb_Switch1 := 1;
        END_IF;

        (* End of Switch: '<S1>/Switch1' *)
        

        (* Outputs for Triggered SubSystem: '<S1>/Subsystem' incorporates:
         *  TriggerPort: '<S2>/Trigger' *)
        i0_ZCFCN_d_FALLING(u0 := Subsystem_Trig_ZCE, u1 := DINT_TO_LREAL(rtb_Switch1));
        tempOutEvent := i0_ZCFCN_d_FALLING.y0;
        Subsystem_Trig_ZCE := i0_ZCFCN_d_FALLING.y1;

        IF tempOutEvent <> 0 THEN 
            (* Inport: '<S2>/pp' *)
            pp := pAsimbar;
            (* Inport: '<S2>/pr' *)
            pr := pBsimbar;
        END_IF;

        (* End of Outputs for SubSystem: '<S1>/Subsystem' *)
        

